LIN {X 0,Y 525.13,Z 398.918,A -85,B 0,C 180,E1 -4783.003,E2 -4783.003} C_VEL
LIN {X 0,Y 525.379,Z 385.467,A -85,B 0,C 180,E1 -4783.44,E2 -4783.44} C_VEL
LIN {X 0,Y 525.572,Z 372.166,A -85,B 0,C 180,E1 -4783.706,E2 -4783.706} C_VEL
LIN {X 0,Y 525.827,Z 279.836,A -85,B 0,C 180,E1 -4784.974,E2 -4784.974} C_VEL
LIN {X 0,Y 524.249,Z 269.867,A -85,B 0,C 180,E1 -4785.172,E2 -4785.172} C_VEL
LIN {X 0,Y 524.68,Z 249.874,A -85,B 0,C 180,E1 -4788.307,E2 -4788.307} C_VEL
LIN {X 0,Y 525.077,Z 230.49,A -85,B 0,C 180,E1 -4791.391,E2 -4791.391} C_VEL
LIN {X 0,Y 525.279,Z 221.566,A -85,B 0,C 180,E1 -4792.831,E2 -4792.831} C_VEL
LIN {X 0,Y 523.919,Z 214.225,A -85,B 0,C 180,E1 -4794.108,E2 -4794.108} C_VEL
LIN {X 0,Y 523.925,Z 214.226,A -85,B 0,C 180,E1 -4797.134,E2 -4797.134} C_VEL
LIN {X 0,Y 523.939,Z 214.222,A -85,B 0,C 180,E1 -4799.756,E2 -4799.756} C_VEL
LIN {X 0,Y 523.935,Z 214.217,A -85,B 0,C 180,E1 -4802.449,E2 -4802.449} C_VEL
LIN {X 0,Y 523.919,Z 214.224,A -85,B 0,C 180,E1 -4805.227,E2 -4805.227} C_VEL
LIN {X 0,Y 523.914,Z 214.221,A -85,B 0,C 180,E1 -4808.102,E2 -4808.102} C_VEL
LIN {X 0,Y 523.938,Z 214.22,A -85,B 0,C 180,E1 -4811.092,E2 -4811.092} C_VEL
LIN {X 0,Y 523.93,Z 214.218,A -85,B 0,C 180,E1 -4814.229,E2 -4814.229} C_VEL
LIN {X 0,Y 523.893,Z 214.223,A -85,B 0,C 180,E1 -4816.83,E2 -4816.83} C_VEL
LIN {X 0,Y 523.938,Z 214.218,A -85,B 0,C 180,E1 -4818.907,E2 -4818.907} C_VEL
LIN {X 0,Y 523.913,Z 214.221,A -85,B 0,C 180,E1 -4821.898,E2 -4821.898} C_VEL
LIN {X 0,Y 523.922,Z 214.22,A -85,B 0,C 180,E1 -4824.912,E2 -4824.912} C_VEL
LIN {X 0,Y 523.936,Z 214.222,A -85,B 0,C 180,E1 -4827.68,E2 -4827.68} C_VEL
LIN {X 0,Y 523.954,Z 214.212,A -85,B 0,C 180,E1 -4830.677,E2 -4830.677} C_VEL
LIN {X 0,Y 523.938,Z 214.219,A -85,B 0,C 180,E1 -4833.727,E2 -4833.727} C_VEL
LIN {X 0,Y 523.913,Z 214.219,A -85,B 0,C 180,E1 -4836.27,E2 -4836.27} C_VEL
LIN {X 0,Y 523.946,Z 214.214,A -85,B 0,C 180,E1 -4838.767,E2 -4838.767} C_VEL
LIN {X 0,Y 523.948,Z 214.221,A -85,B 0,C 180,E1 -4841.221,E2 -4841.221} C_VEL
LIN {X 0,Y 523.928,Z 214.223,A -85,B 0,C 180,E1 -4843.639,E2 -4843.639} C_VEL
LIN {X 0,Y 523.944,Z 214.216,A -85,B 0,C 180,E1 -4846.028,E2 -4846.028} C_VEL
LIN {X 0,Y 523.995,Z 214.212,A -85,B 0,C 180,E1 -4849.177,E2 -4849.177} C_VEL
LIN {X 0,Y 524.029,Z 214.203,A -85,B 0,C 180,E1 -4852.293,E2 -4852.293} C_VEL
LIN {X 0,Y 524.079,Z 214.198,A -85,B 0,C 180,E1 -4854.614,E2 -4854.614} C_VEL
LIN {X 0,Y 524.112,Z 214.197,A -85,B 0,C 180,E1 -4857.695,E2 -4857.695} C_VEL
LIN {X 0,Y 524.119,Z 214.194,A -85,B 0,C 180,E1 -4860.768,E2 -4860.768} C_VEL
LIN {X 0,Y 524.041,Z 214.205,A -85,B 0,C 180,E1 -4863.075,E2 -4863.075} C_VEL
LIN {X 0,Y 524.033,Z 214.204,A -85,B 0,C 180,E1 -4866.159,E2 -4866.159} C_VEL
LIN {X 0,Y 523.985,Z 214.214,A -85,B 0,C 180,E1 -4869.262,E2 -4869.262} C_VEL
LIN {X 0,Y 524.001,Z 214.211,A -85,B 0,C 180,E1 -4871.737,E2 -4871.737} C_VEL
LIN {X 0,Y 523.988,Z 214.212,A -85,B 0,C 180,E1 -4875.05,E2 -4875.05} C_VEL
LIN {X 0,Y 523.946,Z 214.214,A -85,B 0,C 180,E1 -4877.97,E2 -4877.97} C_VEL
LIN {X 0,Y 523.959,Z 214.213,A -85,B 0,C 180,E1 -4880.411,E2 -4880.411} C_VEL
LIN {X 0,Y 523.911,Z 214.219,A -85,B 0,C 180,E1 -4882.894,E2 -4882.894} C_VEL
LIN {X 0,Y 523.911,Z 214.227,A -85,B 0,C 180,E1 -4885.421,E2 -4885.421} C_VEL
LIN {X 0,Y 523.957,Z 214.215,A -85,B 0,C 180,E1 -4888,E2 -4888} C_VEL
LIN {X 0,Y 523.941,Z 214.216,A -85,B 0,C 180,E1 -4890.854,E2 -4890.854} C_VEL
LIN {X 0,Y 523.961,Z 214.218,A -85,B 0,C 180,E1 -4893.734,E2 -4893.734} C_VEL
LIN {X 0,Y 523.9,Z 214.219,A -85,B 0,C 180,E1 -4896.401,E2 -4896.401} C_VEL
LIN {X 0,Y 523.921,Z 214.223,A -85,B 0,C 180,E1 -4899.085,E2 -4899.085} C_VEL
LIN {X 0,Y 523.945,Z 214.216,A -85,B 0,C 180,E1 -4902.12,E2 -4902.12} C_VEL
LIN {X 0,Y 523.94,Z 214.225,A -85,B 0,C 180,E1 -4905.311,E2 -4905.311} C_VEL
LIN {X 0,Y 523.893,Z 214.222,A -85,B 0,C 180,E1 -4906.884,E2 -4906.884} C_VEL
LIN {X 0,Y 523.226,Z 214.314,A -85,B 0,C 180,E1 -4907.526,E2 -4907.526} C_VEL
LIN {X 0,Y 520.369,Z 214.665,A -85,B 0,C 180,E1 -4908.568,E2 -4908.568} C_VEL
LIN {X 0,Y 517.964,Z 214.969,A -85,B 0,C 180,E1 -4909.407,E2 -4909.407} C_VEL
LIN {X 0,Y 516.948,Z 215.089,A -85,B 0,C 180,E1 -4910.055,E2 -4910.055} C_VEL
LIN {X 0,Y 516.873,Z 215.097,A -85,B 0,C 180,E1 -4910.274,E2 -4910.274} C_VEL
LIN {X 0,Y 516.877,Z 215.106,A -85,B 0,C 180,E1 -4913.344,E2 -4913.344} C_VEL
LIN {X 0,Y 516.887,Z 215.096,A -85,B 0,C 180,E1 -4916.119,E2 -4916.119} C_VEL
LIN {X 0,Y 516.894,Z 215.097,A -85,B 0,C 180,E1 -4918.936,E2 -4918.936} C_VEL
LIN {X 0,Y 516.865,Z 215.102,A -85,B 0,C 180,E1 -4921.582,E2 -4921.582} C_VEL
LIN {X 0,Y 516.961,Z 215.274,A -85,B 0,C 180,E1 -4923.533,E2 -4923.533} C_VEL
LIN {X 0,Y 517.58,Z 220.097,A -85,B 0,C 180,E1 -4924.461,E2 -4924.461} C_VEL
LIN {X 0,Y 517.327,Z 236.48,A -85,B 0,C 180,E1 -4927.488,E2 -4927.488} C_VEL
LIN {X 0,Y 517.234,Z 242.99,A -85,B 0,C 180,E1 -4928.68,E2 -4928.68} C_VEL
LIN {X 0,Y 519.15,Z 254.45,A -85,B 0,C 180,E1 -4928.909,E2 -4928.909} C_VEL
LIN {X 0,Y 518.623,Z 349.842,A -85,B 0,C 180,E1 -4930.249,E2 -4930.249} C_VEL
LIN {X 0,Y 518.444,Z 363.428,A -85,B 0,C 180,E1 -4930.602,E2 -4930.602} C_VEL
LIN {X 0,Y 518.199,Z 376.588,A -85,B 0,C 180,E1 -4931.117,E2 -4931.117} C_VEL
LIN {X 0,Y 517.949,Z 388.728,A -85,B 0,C 180,E1 -4931.774,E2 -4931.774} C_VEL
LIN {X 0,Y 517.563,Z 400.832,A -85,B 0,C 180,E1 -4932.618,E2 -4932.618} C_VEL
LIN {X 0,Y 517.292,Z 411.073,A -85,B 0,C 180,E1 -4933.524,E2 -4933.524} C_VEL
LIN {X 0,Y 517.046,Z 419.545,A -85,B 0,C 180,E1 -4934.44,E2 -4934.44} C_VEL
LIN {X 0,Y 516.757,Z 428.512,A -85,B 0,C 180,E1 -4935.629,E2 -4935.629} C_VEL
LIN {X 0,Y 516.583,Z 435.771,A -85,B 0,C 180,E1 -4936.828,E2 -4936.828} C_VEL
LIN {X 0,Y 516.486,Z 440.64,A -85,B 0,C 180,E1 -4937.824,E2 -4937.824} C_VEL
LIN {X 0,Y 516.377,Z 445.343,A -85,B 0,C 180,E1 -4939.016,E2 -4939.016} C_VEL
LIN {X 0,Y 516.282,Z 448.91,A -85,B 0,C 180,E1 -4940.203,E2 -4940.203} C_VEL
LIN {X 0,Y 516.234,Z 451.446,A -85,B 0,C 180,E1 -4941.387,E2 -4941.387} C_VEL
LIN {X 0,Y 516.254,Z 452.623,A -85,B 0,C 180,E1 -4942.176,E2 -4942.176} C_VEL
LIN {X 0,Y 516.273,Z 453.665,A -85,B 0,C 180,E1 -4943.591,E2 -4943.591} C_VEL
LIN {X 0,Y 516.273,Z 453.657,A -85,B 0,C 180,E1 -4944.532,E2 -4944.532} C_VEL
LIN {X 0,Y 516.217,Z 453.229,A -85,B 0,C 180,E1 -4945.314,E2 -4945.314} C_VEL
LIN {X 0,Y 516.304,Z 452.364,A -85,B 0,C 180,E1 -4946.097,E2 -4946.097} C_VEL
LIN {X 0,Y 516.295,Z 451.11,A -85,B 0,C 180,E1 -4946.879,E2 -4946.879} C_VEL
LIN {X 0,Y 516.311,Z 448.459,A -85,B 0,C 180,E1 -4948.05,E2 -4948.05} C_VEL
LIN {X 0,Y 516.283,Z 444.815,A -85,B 0,C 180,E1 -4949.22,E2 -4949.22} C_VEL
LIN {X 0,Y 516.453,Z 440.065,A -85,B 0,C 180,E1 -4950.39,E2 -4950.39} C_VEL
LIN {X 0,Y 516.558,Z 434.09,A -85,B 0,C 180,E1 -4951.559,E2 -4951.559} C_VEL
LIN {X 0,Y 516.82,Z 426.665,A -85,B 0,C 180,E1 -4952.728,E2 -4952.728} C_VEL
LIN {X 0,Y 517.036,Z 419.105,A -85,B 0,C 180,E1 -4953.702,E2 -4953.702} C_VEL
LIN {X 0,Y 517.288,Z 409.943,A -85,B 0,C 180,E1 -4954.676,E2 -4954.676} C_VEL
LIN {X 0,Y 517.632,Z 399.759,A -85,B 0,C 180,E1 -4955.551,E2 -4955.551} C_VEL
LIN {X 0,Y 517.936,Z 388.496,A -85,B 0,C 180,E1 -4956.33,E2 -4956.33} C_VEL
LIN {X 0,Y 518.177,Z 376.803,A -85,B 0,C 180,E1 -4956.962,E2 -4956.962} C_VEL
LIN {X 0,Y 518.46,Z 363.864,A -85,B 0,C 180,E1 -4957.472,E2 -4957.472} C_VEL
LIN {X 0,Y 518.602,Z 351.137,A -85,B 0,C 180,E1 -4957.813,E2 -4957.813} C_VEL
LIN {X 0,Y 518.884,Z 303.338,A -85,B 0,C 180,E1 -4958.501,E2 -4958.501} C_VEL
LIN {X 0,Y 519.104,Z 253.077,A -85,B 0,C 180,E1 -4959.201,E2 -4959.201} C_VEL
LIN {X 0,Y 517.252,Z 243.013,A -85,B 0,C 180,E1 -4959.408,E2 -4959.408} C_VEL
LIN {X 0,Y 517.52,Z 228.477,A -85,B 0,C 180,E1 -4962.102,E2 -4962.102} C_VEL
LIN {X 0,Y 517.546,Z 218.647,A -85,B 0,C 180,E1 -4963.948,E2 -4963.948} C_VEL
LIN {X 0,Y 516.993,Z 215.091,A -85,B 0,C 180,E1 -4964.666,E2 -4964.666} C_VEL
LIN {X 0,Y 516.905,Z 215.095,A -85,B 0,C 180,E1 -4967.871,E2 -4967.871} C_VEL
LIN {X 0,Y 516.916,Z 215.1,A -85,B 0,C 180,E1 -4970.701,E2 -4970.701} C_VEL
LIN {X 0,Y 516.906,Z 215.093,A -85,B 0,C 180,E1 -4974.072,E2 -4974.072} C_VEL
LIN {X 0,Y 516.9,Z 215.101,A -85,B 0,C 180,E1 -4976.659,E2 -4976.659} C_VEL
LIN {X 0,Y 516.913,Z 215.091,A -85,B 0,C 180,E1 -4979.523,E2 -4979.523} C_VEL
LIN {X 0,Y 516.898,Z 215.1,A -85,B 0,C 180,E1 -4982.543,E2 -4982.543} C_VEL
LIN {X 0,Y 516.866,Z 215.098,A -85,B 0,C 180,E1 -4985.329,E2 -4985.329} C_VEL
LIN {X 0,Y 516.881,Z 215.095,A -85,B 0,C 180,E1 -4987.943,E2 -4987.943} C_VEL
LIN {X 0,Y 516.885,Z 215.103,A -85,B 0,C 180,E1 -4990.742,E2 -4990.742} C_VEL
LIN {X 0,Y 516.884,Z 215.101,A -85,B 0,C 180,E1 -4992.831,E2 -4992.831} C_VEL
LIN {X 0,Y 516.897,Z 215.097,A -85,B 0,C 180,E1 -4995.007,E2 -4995.007} C_VEL
LIN {X 0,Y 516.912,Z 215.096,A -85,B 0,C 180,E1 -4998.399,E2 -4998.399} C_VEL
LIN {X 0,Y 516.881,Z 215.096,A -85,B 0,C 180,E1 -5001.284,E2 -5001.284} C_VEL
LIN {X 0,Y 516.869,Z 215.099,A -85,B 0,C 180,E1 -5004.219,E2 -5004.219} C_VEL
LIN {X 0,Y 516.896,Z 215.096,A -85,B 0,C 180,E1 -5007.053,E2 -5007.053} C_VEL
LIN {X 0,Y 516.893,Z 215.093,A -85,B 0,C 180,E1 -5009.796,E2 -5009.796} C_VEL
LIN {X 0,Y 516.922,Z 215.096,A -85,B 0,C 180,E1 -5012.467,E2 -5012.467} C_VEL
LIN {X 0,Y 516.877,Z 215.095,A -85,B 0,C 180,E1 -5015.644,E2 -5015.644} C_VEL
LIN {X 0,Y 516.887,Z 215.101,A -85,B 0,C 180,E1 -5018.462,E2 -5018.462} C_VEL
LIN {X 0,Y 516.895,Z 215.097,A -85,B 0,C 180,E1 -5020.954,E2 -5020.954} C_VEL
LIN {X 0,Y 516.901,Z 215.092,A -85,B 0,C 180,E1 -5023.41,E2 -5023.41} C_VEL
LIN {X 0,Y 516.885,Z 215.094,A -85,B 0,C 180,E1 -5025.833,E2 -5025.833} C_VEL
LIN {X 0,Y 516.951,Z 215.089,A -85,B 0,C 180,E1 -5029.028,E2 -5029.028} C_VEL
LIN {X 0,Y 516.963,Z 215.087,A -85,B 0,C 180,E1 -5032.186,E2 -5032.186} C_VEL
LIN {X 0,Y 517.025,Z 215.085,A -85,B 0,C 180,E1 -5034.54,E2 -5034.54} C_VEL
LIN {X 0,Y 517.083,Z 215.069,A -85,B 0,C 180,E1 -5037.663,E2 -5037.663} C_VEL
LIN {X 0,Y 517.093,Z 215.075,A -85,B 0,C 180,E1 -5040.779,E2 -5040.779} C_VEL
LIN {X 0,Y 516.985,Z 215.084,A -85,B 0,C 180,E1 -5043.117,E2 -5043.117} C_VEL
LIN {X 0,Y 517.009,Z 215.083,A -85,B 0,C 180,E1 -5046.243,E2 -5046.243} C_VEL
LIN {X 0,Y 516.943,Z 215.087,A -85,B 0,C 180,E1 -5049.389,E2 -5049.389} C_VEL
LIN {X 0,Y 516.953,Z 215.086,A -85,B 0,C 180,E1 -5051.807,E2 -5051.807} C_VEL
LIN {X 0,Y 516.948,Z 215.088,A -85,B 0,C 180,E1 -5055.148,E2 -5055.148} C_VEL
LIN {X 0,Y 516.916,Z 215.094,A -85,B 0,C 180,E1 -5058.223,E2 -5058.223} C_VEL
LIN {X 0,Y 516.913,Z 215.098,A -85,B 0,C 180,E1 -5060.701,E2 -5060.701} C_VEL
LIN {X 0,Y 516.903,Z 215.094,A -85,B 0,C 180,E1 -5064.072,E2 -5064.072} C_VEL
LIN {X 0,Y 516.897,Z 215.101,A -85,B 0,C 180,E1 -5066.659,E2 -5066.659} C_VEL
LIN {X 0,Y 516.91,Z 215.091,A -85,B 0,C 180,E1 -5069.523,E2 -5069.523} C_VEL
LIN {X 0,Y 516.895,Z 215.102,A -85,B 0,C 180,E1 -5072.543,E2 -5072.543} C_VEL
LIN {X 0,Y 516.864,Z 215.097,A -85,B 0,C 180,E1 -5075.329,E2 -5075.329} C_VEL
LIN {X 0,Y 516.879,Z 215.096,A -85,B 0,C 180,E1 -5077.943,E2 -5077.943} C_VEL
LIN {X 0,Y 516.882,Z 215.101,A -85,B 0,C 180,E1 -5080.742,E2 -5080.742} C_VEL
LIN {X 0,Y 516.881,Z 215.096,A -85,B 0,C 180,E1 -5083.903,E2 -5083.903} C_VEL
LIN {X 0,Y 516.882,Z 215.098,A -85,B 0,C 180,E1 -5086.107,E2 -5086.107} C_VEL
LIN {X 0,Y 516.883,Z 215.095,A -85,B 0,C 180,E1 -5089.258,E2 -5089.258} C_VEL
LIN {X 0,Y 516.861,Z 215.102,A -85,B 0,C 180,E1 -5092.274,E2 -5092.274} C_VEL
LIN {X 0,Y 516.883,Z 215.096,A -85,B 0,C 180,E1 -5095.175,E2 -5095.175} C_VEL
LIN {X 0,Y 516.875,Z 215.097,A -85,B 0,C 180,E1 -5097.975,E2 -5097.975} C_VEL
LIN {X 0,Y 516.922,Z 215.097,A -85,B 0,C 180,E1 -5100.696,E2 -5100.696} C_VEL
LIN {X 0,Y 516.905,Z 215.095,A -85,B 0,C 180,E1 -5103.341,E2 -5103.341} C_VEL
LIN {X 0,Y 516.908,Z 215.177,A -85,B 0,C 180,E1 -5105.752,E2 -5105.752} C_VEL
LIN {X 0,Y 518.35,Z 223.667,A -85,B 0,C 180,E1 -5107.217,E2 -5107.217} C_VEL
LIN {X 0,Y 517.938,Z 240.677,A -85,B 0,C 180,E1 -5109.979,E2 -5109.979} C_VEL
LIN {X 0,Y 517.486,Z 258.383,A -85,B 0,C 180,E1 -5112.819,E2 -5112.819} C_VEL
LIN {X 0,Y 517.275,Z 269.968,A -85,B 0,C 180,E1 -5114.636,E2 -5114.636} C_VEL
LIN {X 0,Y 519.06,Z 282.453,A -85,B 0,C 180,E1 -5114.865,E2 -5114.865} C_VEL
LIN {X 0,Y 518.609,Z 377.87,A -85,B 0,C 180,E1 -5116.206,E2 -5116.206} C_VEL
LIN {X 0,Y 518.373,Z 391.174,A -85,B 0,C 180,E1 -5116.55,E2 -5116.55} C_VEL
LIN {X 0,Y 518.092,Z 403.355,A -85,B 0,C 180,E1 -5117.016,E2 -5117.016} C_VEL
LIN {X 0,Y 517.768,Z 415.713,A -85,B 0,C 180,E1 -5117.66,E2 -5117.66} C_VEL
LIN {X 0,Y 517.554,Z 427.254,A -85,B 0,C 180,E1 -5118.446,E2 -5118.446} C_VEL
LIN {X 0,Y 517.22,Z 437.703,A -85,B 0,C 180,E1 -5119.331,E2 -5119.331} C_VEL
LIN {X 0,Y 516.95,Z 446.247,A -85,B 0,C 180,E1 -5120.216,E2 -5120.216} C_VEL
LIN {X 0,Y 516.724,Z 454.13,A -85,B 0,C 180,E1 -5121.199,E2 -5121.199} C_VEL
LIN {X 0,Y 516.536,Z 461.829,A -85,B 0,C 180,E1 -5122.377,E2 -5122.377} C_VEL
LIN {X 0,Y 516.39,Z 468.926,A -85,B 0,C 180,E1 -5123.749,E2 -5123.749} C_VEL
LIN {X 0,Y 516.313,Z 473.647,A -85,B 0,C 180,E1 -5124.924,E2 -5124.924} C_VEL
LIN {X 0,Y 516.352,Z 477.256,A -85,B 0,C 180,E1 -5126.098,E2 -5126.098} C_VEL
LIN {X 0,Y 516.282,Z 479.114,A -85,B 0,C 180,E1 -5126.879,E2 -5126.879} C_VEL
LIN {X 0,Y 516.261,Z 480.509,A -85,B 0,C 180,E1 -5127.659,E2 -5127.659} C_VEL
LIN {X 0,Y 516.161,Z 482.109,A -85,B 0,C 180,E1 -5129.22,E2 -5129.22} C_VEL
LIN {X 0,Y 516.157,Z 482.324,A -85,B 0,C 180,E1 -5130,E2 -5130} C_VEL
LIN {X 0,Y 516.192,Z 481.502,A -85,B 0,C 180,E1 -5131.56,E2 -5131.56} C_VEL
LIN {X 0,Y 516.261,Z 480.508,A -85,B 0,C 180,E1 -5132.341,E2 -5132.341} C_VEL
LIN {X 0,Y 516.282,Z 479.113,A -85,B 0,C 180,E1 -5133.121,E2 -5133.121} C_VEL
LIN {X 0,Y 516.311,Z 476.179,A -85,B 0,C 180,E1 -5134.294,E2 -5134.294} C_VEL
LIN {X 0,Y 516.374,Z 472.206,A -85,B 0,C 180,E1 -5135.467,E2 -5135.467} C_VEL
LIN {X 0,Y 516.422,Z 467.014,A -85,B 0,C 180,E1 -5136.659,E2 -5136.659} C_VEL
LIN {X 0,Y 516.575,Z 460.656,A -85,B 0,C 180,E1 -5137.819,E2 -5137.819} C_VEL
LIN {X 0,Y 516.769,Z 452.625,A -85,B 0,C 180,E1 -5138.998,E2 -5138.998} C_VEL
LIN {X 0,Y 516.98,Z 444.442,A -85,B 0,C 180,E1 -5139.981,E2 -5139.981} C_VEL
LIN {X 0,Y 517.331,Z 434.466,A -85,B 0,C 180,E1 -5140.964,E2 -5140.964} C_VEL
LIN {X 0,Y 517.604,Z 424.623,A -85,B 0,C 180,E1 -5141.752,E2 -5141.752} C_VEL
LIN {X 0,Y 517.849,Z 413.514,A -85,B 0,C 180,E1 -5142.465,E2 -5142.465} C_VEL
LIN {X 0,Y 518.132,Z 401.058,A -85,B 0,C 180,E1 -5143.082,E2 -5143.082} C_VEL
LIN {X 0,Y 518.442,Z 388.005,A -85,B 0,C 180,E1 -5143.548,E2 -5143.548} C_VEL
LIN {X 0,Y 518.629,Z 374.978,A -85,B 0,C 180,E1 -5143.843,E2 -5143.843} C_VEL
LIN {X 0,Y 518.989,Z 280.748,A -85,B 0,C 180,E1 -5145.16,E2 -5145.16} C_VEL
LIN {X 0,Y 517.238,Z 269.601,A -85,B 0,C 180,E1 -5145.393,E2 -5145.393} C_VEL
LIN {X 0,Y 517.721,Z 249.417,A -85,B 0,C 180,E1 -5148.603,E2 -5148.603} C_VEL
LIN {X 0,Y 518.132,Z 231.593,A -85,B 0,C 180,E1 -5151.483,E2 -5151.483} C_VEL
LIN {X 0,Y 518.327,Z 222.878,A -85,B 0,C 180,E1 -5152.912,E2 -5152.912} C_VEL
LIN {X 0,Y 516.899,Z 215.098,A -85,B 0,C 180,E1 -5154.314,E2 -5154.314} C_VEL
LIN {X 0,Y 516.901,Z 215.102,A -85,B 0,C 180,E1 -5157.534,E2 -5157.534} C_VEL
LIN {X 0,Y 516.888,Z 215.096,A -85,B 0,C 180,E1 -5160.204,E2 -5160.204} C_VEL
LIN {X 0,Y 516.897,Z 215.096,A -85,B 0,C 180,E1 -5162.947,E2 -5162.947} C_VEL
LIN {X 0,Y 516.869,Z 215.102,A -85,B 0,C 180,E1 -5165.781,E2 -5165.781} C_VEL
LIN {X 0,Y 516.88,Z 215.096,A -85,B 0,C 180,E1 -5168.716,E2 -5168.716} C_VEL
LIN {X 0,Y 516.908,Z 215.097,A -85,B 0,C 180,E1 -5171.776,E2 -5171.776} C_VEL
LIN {X 0,Y 516.896,Z 215.096,A -85,B 0,C 180,E1 -5175.007,E2 -5175.007} C_VEL
LIN {X 0,Y 516.91,Z 215.092,A -85,B 0,C 180,E1 -5178.399,E2 -5178.399} C_VEL
LIN {X 0,Y 516.877,Z 215.102,A -85,B 0,C 180,E1 -5181.284,E2 -5181.284} C_VEL
LIN {X 0,Y 516.867,Z 215.097,A -85,B 0,C 180,E1 -5184.219,E2 -5184.219} C_VEL
LIN {X 0,Y 516.882,Z 215.096,A -85,B 0,C 180,E1 -5187.052,E2 -5187.052} C_VEL
LIN {X 0,Y 516.892,Z 215.095,A -85,B 0,C 180,E1 -5189.796,E2 -5189.796} C_VEL
LIN {X 0,Y 516.898,Z 215.093,A -85,B 0,C 180,E1 -5192.466,E2 -5192.466} C_VEL
LIN {X 0,Y 516.867,Z 215.098,A -85,B 0,C 180,E1 -5195.07,E2 -5195.07} C_VEL
LIN {X 0,Y 516.87,Z 215.101,A -85,B 0,C 180,E1 -5197.622,E2 -5197.622} C_VEL
LIN {X 0,Y 516.932,Z 215.089,A -85,B 0,C 180,E1 -5200.13,E2 -5200.13} C_VEL
LIN {X 0,Y 516.906,Z 215.091,A -85,B 0,C 180,E1 -5202.595,E2 -5202.595} C_VEL
LIN {X 0,Y 516.953,Z 215.089,A -85,B 0,C 180,E1 -5205.03,E2 -5205.03} C_VEL
LIN {X 0,Y 516.967,Z 215.082,A -85,B 0,C 180,E1 -5208.234,E2 -5208.234} C_VEL
LIN {X 0,Y 516.965,Z 215.093,A -85,B 0,C 180,E1 -5211.4,E2 -5211.4} C_VEL
LIN {X 0,Y 517.009,Z 215.083,A -85,B 0,C 180,E1 -5213.757,E2 -5213.757} C_VEL
LIN {X 0,Y 517.082,Z 215.073,A -85,B 0,C 180,E1 -5217.663,E2 -5217.663} C_VEL
LIN {X 0,Y 517.09,Z 215.07,A -85,B 0,C 180,E1 -5220.779,E2 -5220.779} C_VEL
LIN {X 0,Y 516.984,Z 215.085,A -85,B 0,C 180,E1 -5223.117,E2 -5223.117} C_VEL
LIN {X 0,Y 516.995,Z 215.081,A -85,B 0,C 180,E1 -5226.243,E2 -5226.243} C_VEL
LIN {X 0,Y 516.941,Z 215.093,A -85,B 0,C 180,E1 -5229.39,E2 -5229.39} C_VEL
LIN {X 0,Y 516.953,Z 215.088,A -85,B 0,C 180,E1 -5231.807,E2 -5231.807} C_VEL
LIN {X 0,Y 516.94,Z 215.091,A -85,B 0,C 180,E1 -5235.144,E2 -5235.144} C_VEL
LIN {X 0,Y 516.914,Z 215.088,A -85,B 0,C 180,E1 -5238.223,E2 -5238.223} C_VEL
LIN {X 0,Y 516.906,Z 215.092,A -85,B 0,C 180,E1 -5240.702,E2 -5240.702} C_VEL
LIN {X 0,Y 516.887,Z 215.095,A -85,B 0,C 180,E1 -5244.073,E2 -5244.073} C_VEL
LIN {X 0,Y 516.905,Z 215.09,A -85,B 0,C 180,E1 -5246.659,E2 -5246.659} C_VEL
LIN {X 0,Y 516.91,Z 215.097,A -85,B 0,C 180,E1 -5249.523,E2 -5249.523} C_VEL
LIN {X 0,Y 516.897,Z 215.093,A -85,B 0,C 180,E1 -5252.543,E2 -5252.543} C_VEL
LIN {X 0,Y 516.866,Z 215.105,A -85,B 0,C 180,E1 -5255.329,E2 -5255.329} C_VEL
LIN {X 0,Y 516.88,Z 215.097,A -85,B 0,C 180,E1 -5257.943,E2 -5257.943} C_VEL
LIN {X 0,Y 516.884,Z 215.096,A -85,B 0,C 180,E1 -5260.742,E2 -5260.742} C_VEL
LIN {X 0,Y 516.883,Z 215.098,A -85,B 0,C 180,E1 -5263.903,E2 -5263.903} C_VEL
LIN {X 0,Y 516.846,Z 215.1,A -85,B 0,C 180,E1 -5266.886,E2 -5266.886} C_VEL
LIN {X 0,Y 516.886,Z 215.101,A -85,B 0,C 180,E1 -5269.59,E2 -5269.59} C_VEL
LIN {X 0,Y 516.873,Z 215.097,A -85,B 0,C 180,E1 -5270.274,E2 -5270.274} C_VEL
LIN {X 0,Y 516.232,Z 215.18,A -85,B 0,C 180,E1 -5270.924,E2 -5270.924} C_VEL
LIN {X 0,Y 513.391,Z 215.54,A -85,B 0,C 180,E1 -5271.98,E2 -5271.98} C_VEL
LIN {X 0,Y 510.967,Z 215.845,A -85,B 0,C 180,E1 -5272.83,E2 -5272.83} C_VEL
LIN {X 0,Y 509.913,Z 215.973,A -85,B 0,C 180,E1 -5273.487,E2 -5273.487} C_VEL
LIN {X 0,Y 509.822,Z 215.982,A -85,B 0,C 180,E1 -5273.709,E2 -5273.709} C_VEL
LIN {X 0,Y 509.844,Z 215.973,A -85,B 0,C 180,E1 -5276.538,E2 -5276.538} C_VEL
LIN {X 0,Y 509.848,Z 215.978,A -85,B 0,C 180,E1 -5279.334,E2 -5279.334} C_VEL
LIN {X 0,Y 509.851,Z 215.974,A -85,B 0,C 180,E1 -5282.052,E2 -5282.052} C_VEL
LIN {X 0,Y 509.904,Z 216.009,A -85,B 0,C 180,E1 -5283.361,E2 -5283.361} C_VEL
LIN {X 0,Y 510.626,Z 221.981,A -85,B 0,C 180,E1 -5284.525,E2 -5284.525} C_VEL
LIN {X 0,Y 510.333,Z 238.095,A -85,B 0,C 180,E1 -5287.533,E2 -5287.533} C_VEL
LIN {X 0,Y 510.273,Z 243.432,A -85,B 0,C 180,E1 -5288.477,E2 -5288.477} C_VEL
LIN {X 0,Y 512.315,Z 255.262,A -85,B 0,C 180,E1 -5288.711,E2 -5288.711} C_VEL
LIN {X 0,Y 511.732,Z 350.795,A -85,B 0,C 180,E1 -5290.076,E2 -5290.076} C_VEL
LIN {X 0,Y 511.546,Z 364.127,A -85,B 0,C 180,E1 -5290.435,E2 -5290.435} C_VEL
LIN {X 0,Y 511.293,Z 376.918,A -85,B 0,C 180,E1 -5290.946,E2 -5290.946} C_VEL
LIN {X 0,Y 511.017,Z 389.089,A -85,B 0,C 180,E1 -5291.615,E2 -5291.615} C_VEL
LIN {X 0,Y 510.643,Z 399.924,A -85,B 0,C 180,E1 -5292.375,E2 -5292.375} C_VEL
LIN {X 0,Y 510.358,Z 410.422,A -85,B 0,C 180,E1 -5293.294,E2 -5293.294} C_VEL
LIN {X 0,Y 510.047,Z 418.946,A -85,B 0,C 180,E1 -5294.209,E2 -5294.209} C_VEL
LIN {X 0,Y 509.742,Z 428.132,A -85,B 0,C 180,E1 -5295.427,E2 -5295.427} C_VEL
LIN {X 0,Y 509.524,Z 435.499,A -85,B 0,C 180,E1 -5296.642,E2 -5296.642} C_VEL
LIN {X 0,Y 509.417,Z 440.453,A -85,B 0,C 180,E1 -5297.652,E2 -5297.652} C_VEL
LIN {X 0,Y 509.325,Z 445.239,A -85,B 0,C 180,E1 -5298.861,E2 -5298.861} C_VEL
LIN {X 0,Y 509.222,Z 448.882,A -85,B 0,C 180,E1 -5300.066,E2 -5300.066} C_VEL
LIN {X 0,Y 509.145,Z 451.49,A -85,B 0,C 180,E1 -5301.266,E2 -5301.266} C_VEL
LIN {X 0,Y 509.163,Z 452.712,A -85,B 0,C 180,E1 -5302.066,E2 -5302.066} C_VEL
LIN {X 0,Y 509.2,Z 453.5,A -85,B 0,C 180,E1 -5302.864,E2 -5302.864} C_VEL
LIN {X 0,Y 509.182,Z 453.87,A -85,B 0,C 180,E1 -5304.456,E2 -5304.456} C_VEL
LIN {X 0,Y 509.133,Z 453.484,A -85,B 0,C 180,E1 -5305.249,E2 -5305.249} C_VEL
LIN {X 0,Y 509.198,Z 452.677,A -85,B 0,C 180,E1 -5306.043,E2 -5306.043} C_VEL
LIN {X 0,Y 509.209,Z 451.457,A -85,B 0,C 180,E1 -5306.835,E2 -5306.835} C_VEL
LIN {X 0,Y 509.22,Z 448.876,A -85,B 0,C 180,E1 -5308.023,E2 -5308.023} C_VEL
LIN {X 0,Y 509.199,Z 445.306,A -85,B 0,C 180,E1 -5309.209,E2 -5309.209} C_VEL
LIN {X 0,Y 509.371,Z 440.636,A -85,B 0,C 180,E1 -5310.395,E2 -5310.395} C_VEL
LIN {X 0,Y 509.493,Z 434.747,A -85,B 0,C 180,E1 -5311.581,E2 -5311.581} C_VEL
LIN {X 0,Y 509.667,Z 428.764,A -85,B 0,C 180,E1 -5312.569,E2 -5312.569} C_VEL
LIN {X 0,Y 509.981,Z 419.975,A -85,B 0,C 180,E1 -5313.753,E2 -5313.753} C_VEL
LIN {X 0,Y 510.272,Z 410.978,A -85,B 0,C 180,E1 -5314.74,E2 -5314.74} C_VEL
LIN {X 0,Y 510.619,Z 401.022,A -85,B 0,C 180,E1 -5315.628,E2 -5315.628} C_VEL
LIN {X 0,Y 510.97,Z 389.991,A -85,B 0,C 180,E1 -5316.416,E2 -5316.416} C_VEL
LIN {X 0,Y 511.258,Z 377.66,A -85,B 0,C 180,E1 -5317.107,E2 -5317.107} C_VEL
LIN {X 0,Y 511.548,Z 365.063,A -85,B 0,C 180,E1 -5317.624,E2 -5317.624} C_VEL
LIN {X 0,Y 511.743,Z 351.073,A -85,B 0,C 180,E1 -5318.007,E2 -5318.007} C_VEL
LIN {X 0,Y 512.208,Z 271.294,A -85,B 0,C 180,E1 -5319.153,E2 -5319.153} C_VEL
LIN {X 0,Y 512.169,Z 253.423,A -85,B 0,C 180,E1 -5319.409,E2 -5319.409} C_VEL
LIN {X 0,Y 510.23,Z 243.085,A -85,B 0,C 180,E1 -5319.639,E2 -5319.639} C_VEL
LIN {X 0,Y 510.519,Z 229.373,A -85,B 0,C 180,E1 -5322.199,E2 -5322.199} C_VEL
LIN {X 0,Y 510.614,Z 220.177,A -85,B 0,C 180,E1 -5323.938,E2 -5323.938} C_VEL
LIN {X 0,Y 509.942,Z 215.969,A -85,B 0,C 180,E1 -5324.772,E2 -5324.772} C_VEL
LIN {X 0,Y 509.871,Z 215.971,A -85,B 0,C 180,E1 -5327.993,E2 -5327.993} C_VEL
LIN {X 0,Y 509.89,Z 215.97,A -85,B 0,C 180,E1 -5330.401,E2 -5330.401} C_VEL
LIN {X 0,Y 509.833,Z 215.973,A -85,B 0,C 180,E1 -5333.563,E2 -5333.563} C_VEL
LIN {X 0,Y 509.882,Z 215.971,A -85,B 0,C 180,E1 -5336.371,E2 -5336.371} C_VEL
LIN {X 0,Y 509.861,Z 215.969,A -85,B 0,C 180,E1 -5339.726,E2 -5339.726} C_VEL
LIN {X 0,Y 509.876,Z 215.975,A -85,B 0,C 180,E1 -5342.774,E2 -5342.774} C_VEL
LIN {X 0,Y 509.826,Z 215.974,A -85,B 0,C 180,E1 -5345.578,E2 -5345.578} C_VEL
LIN {X 0,Y 509.851,Z 215.975,A -85,B 0,C 180,E1 -5348.338,E2 -5348.338} C_VEL
LIN {X 0,Y 509.857,Z 215.97,A -85,B 0,C 180,E1 -5351.425,E2 -5351.425} C_VEL
LIN {X 0,Y 509.841,Z 215.981,A -85,B 0,C 180,E1 -5354.67,E2 -5354.67} C_VEL
LIN {X 0,Y 509.852,Z 215.972,A -85,B 0,C 180,E1 -5358.104,E2 -5358.104} C_VEL
LIN {X 0,Y 509.847,Z 215.98,A -85,B 0,C 180,E1 -5360.647,E2 -5360.647} C_VEL
LIN {X 0,Y 509.81,Z 215.975,A -85,B 0,C 180,E1 -5363.645,E2 -5363.645} C_VEL
LIN {X 0,Y 509.86,Z 215.977,A -85,B 0,C 180,E1 -5366.539,E2 -5366.539} C_VEL
LIN {X 0,Y 509.847,Z 215.972,A -85,B 0,C 180,E1 -5369.334,E2 -5369.334} C_VEL
LIN {X 0,Y 509.884,Z 215.968,A -85,B 0,C 180,E1 -5372.054,E2 -5372.054} C_VEL
LIN {X 0,Y 509.81,Z 215.984,A -85,B 0,C 180,E1 -5374.7,E2 -5374.7} C_VEL
LIN {X 0,Y 509.827,Z 215.974,A -85,B 0,C 180,E1 -5377.458,E2 -5377.458} C_VEL
LIN {X 0,Y 509.917,Z 215.962,A -85,B 0,C 180,E1 -5379.845,E2 -5379.845} C_VEL
LIN {X 0,Y 509.868,Z 215.97,A -85,B 0,C 180,E1 -5383.174,E2 -5383.174} C_VEL
LIN {X 0,Y 509.856,Z 215.97,A -85,B 0,C 180,E1 -5385.634,E2 -5385.634} C_VEL
LIN {X 0,Y 509.913,Z 215.968,A -85,B 0,C 180,E1 -5388.874,E2 -5388.874} C_VEL
LIN {X 0,Y 509.922,Z 215.964,A -85,B 0,C 180,E1 -5392.078,E2 -5392.078} C_VEL
LIN {X 0,Y 509.976,Z 215.962,A -85,B 0,C 180,E1 -5394.464,E2 -5394.464} C_VEL
LIN {X 0,Y 510.054,Z 215.945,A -85,B 0,C 180,E1 -5397.631,E2 -5397.631} C_VEL
LIN {X 0,Y 510.063,Z 215.95,A -85,B 0,C 180,E1 -5400.789,E2 -5400.789} C_VEL
LIN {X 0,Y 509.928,Z 215.963,A -85,B 0,C 180,E1 -5403.16,E2 -5403.16} C_VEL
LIN {X 0,Y 509.977,Z 215.96,A -85,B 0,C 180,E1 -5406.33,E2 -5406.33} C_VEL
LIN {X 0,Y 509.911,Z 215.97,A -85,B 0,C 180,E1 -5408.72,E2 -5408.72} C_VEL
LIN {X 0,Y 509.905,Z 215.965,A -85,B 0,C 180,E1 -5411.932,E2 -5411.932} C_VEL
LIN {X 0,Y 509.895,Z 215.966,A -85,B 0,C 180,E1 -5415.242,E2 -5415.242} C_VEL
LIN {X 0,Y 509.861,Z 215.977,A -85,B 0,C 180,E1 -5418.484,E2 -5418.484} C_VEL
LIN {X 0,Y 509.851,Z 215.974,A -85,B 0,C 180,E1 -5421.002,E2 -5421.002} C_VEL
LIN {X 0,Y 509.858,Z 215.976,A -85,B 0,C 180,E1 -5424.427,E2 -5424.427} C_VEL
LIN {X 0,Y 509.859,Z 215.972,A -85,B 0,C 180,E1 -5427.057,E2 -5427.057} C_VEL
LIN {X 0,Y 509.858,Z 215.97,A -85,B 0,C 180,E1 -5429.751,E2 -5429.751} C_VEL
LIN {X 0,Y 509.867,Z 215.974,A -85,B 0,C 180,E1 -5432.773,E2 -5432.773} C_VEL
LIN {X 0,Y 509.823,Z 215.974,A -85,B 0,C 180,E1 -5435.578,E2 -5435.578} C_VEL
LIN {X 0,Y 509.849,Z 215.976,A -85,B 0,C 180,E1 -5438.338,E2 -5438.338} C_VEL
LIN {X 0,Y 509.853,Z 215.97,A -85,B 0,C 180,E1 -5441.426,E2 -5441.426} C_VEL
LIN {X 0,Y 509.839,Z 215.979,A -85,B 0,C 180,E1 -5444.67,E2 -5444.67} C_VEL
LIN {X 0,Y 509.851,Z 215.973,A -85,B 0,C 180,E1 -5448.104,E2 -5448.104} C_VEL
LIN {X 0,Y 509.846,Z 215.979,A -85,B 0,C 180,E1 -5450.648,E2 -5450.648} C_VEL
LIN {X 0,Y 509.81,Z 215.976,A -85,B 0,C 180,E1 -5453.646,E2 -5453.646} C_VEL
LIN {X 0,Y 509.86,Z 215.979,A -85,B 0,C 180,E1 -5456.539,E2 -5456.539} C_VEL
LIN {X 0,Y 509.844,Z 215.972,A -85,B 0,C 180,E1 -5459.334,E2 -5459.334} C_VEL
LIN {X 0,Y 509.884,Z 215.971,A -85,B 0,C 180,E1 -5462.054,E2 -5462.054} C_VEL
LIN {X 0,Y 509.81,Z 215.981,A -85,B 0,C 180,E1 -5464.7,E2 -5464.7} C_VEL
LIN {X 0,Y 509.869,Z 216.109,A -85,B 0,C 180,E1 -5465.601,E2 -5465.601} C_VEL
LIN {X 0,Y 511.38,Z 224.33,A -85,B 0,C 180,E1 -5467.043,E2 -5467.043} C_VEL
LIN {X 0,Y 510.999,Z 239.669,A -85,B 0,C 180,E1 -5469.567,E2 -5469.567} C_VEL
LIN {X 0,Y 510.536,Z 256.913,A -85,B 0,C 180,E1 -5472.371,E2 -5472.371} C_VEL
LIN {X 0,Y 510.236,Z 269.588,A -85,B 0,C 180,E1 -5474.415,E2 -5474.415} C_VEL
LIN {X 0,Y 512.148,Z 281.846,A -85,B 0,C 180,E1 -5474.65,E2 -5474.65} C_VEL
LIN {X 0,Y 511.726,Z 377.664,A -85,B 0,C 180,E1 -5476.017,E2 -5476.017} C_VEL
LIN {X 0,Y 511.477,Z 390.971,A -85,B 0,C 180,E1 -5476.365,E2 -5476.365} C_VEL
LIN {X 0,Y 511.159,Z 403.154,A -85,B 0,C 180,E1 -5476.837,E2 -5476.837} C_VEL
LIN {X 0,Y 510.872,Z 414.68,A -85,B 0,C 180,E1 -5477.439,E2 -5477.439} C_VEL
LIN {X 0,Y 510.592,Z 425.759,A -85,B 0,C 180,E1 -5478.185,E2 -5478.185} C_VEL
LIN {X 0,Y 510.266,Z 436.433,A -85,B 0,C 180,E1 -5479.083,E2 -5479.083} C_VEL
LIN {X 0,Y 509.916,Z 446.049,A -85,B 0,C 180,E1 -5480.079,E2 -5480.079} C_VEL
LIN {X 0,Y 509.672,Z 453.932,A -85,B 0,C 180,E1 -5481.076,E2 -5481.076} C_VEL
LIN {X 0,Y 509.475,Z 461.632,A -85,B 0,C 180,E1 -5482.27,E2 -5482.27} C_VEL
LIN {X 0,Y 509.308,Z 468.729,A -85,B 0,C 180,E1 -5483.662,E2 -5483.662} C_VEL
LIN {X 0,Y 509.243,Z 473.451,A -85,B 0,C 180,E1 -5484.853,E2 -5484.853} C_VEL
LIN {X 0,Y 509.245,Z 477.059,A -85,B 0,C 180,E1 -5486.043,E2 -5486.043} C_VEL
LIN {X 0,Y 509.2,Z 478.919,A -85,B 0,C 180,E1 -5486.835,E2 -5486.835} C_VEL
LIN {X 0,Y 509.19,Z 480.313,A -85,B 0,C 180,E1 -5487.627,E2 -5487.627} C_VEL
LIN {X 0,Y 509.074,Z 481.913,A -85,B 0,C 180,E1 -5489.209,E2 -5489.209} C_VEL
LIN {X 0,Y 509.068,Z 482.128,A -85,B 0,C 180,E1 -5490,E2 -5490} C_VEL
LIN {X 0,Y 509.112,Z 481.305,A -85,B 0,C 180,E1 -5491.582,E2 -5491.582} C_VEL
LIN {X 0,Y 509.19,Z 480.312,A -85,B 0,C 180,E1 -5492.373,E2 -5492.373} C_VEL
LIN {X 0,Y 509.2,Z 478.916,A -85,B 0,C 180,E1 -5493.165,E2 -5493.165} C_VEL
LIN {X 0,Y 509.203,Z 475.98,A -85,B 0,C 180,E1 -5494.354,E2 -5494.354} C_VEL
LIN {X 0,Y 509.291,Z 472.007,A -85,B 0,C 180,E1 -5495.543,E2 -5495.543} C_VEL
LIN {X 0,Y 509.4,Z 465.998,A -85,B 0,C 180,E1 -5496.914,E2 -5496.914} C_VEL
LIN {X 0,Y 509.545,Z 459.218,A -85,B 0,C 180,E1 -5498.127,E2 -5498.127} C_VEL
LIN {X 0,Y 509.748,Z 450.931,A -85,B 0,C 180,E1 -5499.323,E2 -5499.323} C_VEL
LIN {X 0,Y 510.011,Z 442.439,A -85,B 0,C 180,E1 -5500.32,E2 -5500.32} C_VEL
LIN {X 0,Y 510.382,Z 431.946,A -85,B 0,C 180,E1 -5501.316,E2 -5501.316} C_VEL
LIN {X 0,Y 510.675,Z 421.767,A -85,B 0,C 180,E1 -5502.101,E2 -5502.101} C_VEL
LIN {X 0,Y 511.022,Z 410.185,A -85,B 0,C 180,E1 -5502.813,E2 -5502.813} C_VEL
LIN {X 0,Y 511.293,Z 398.505,A -85,B 0,C 180,E1 -5503.362,E2 -5503.362} C_VEL
LIN {X 0,Y 511.57,Z 385.049,A -85,B 0,C 180,E1 -5503.81,E2 -5503.81} C_VEL
LIN {X 0,Y 511.789,Z 371.734,A -85,B 0,C 180,E1 -5504.082,E2 -5504.082} C_VEL
LIN {X 0,Y 512.108,Z 281.456,A -85,B 0,C 180,E1 -5505.356,E2 -5505.356} C_VEL
LIN {X 0,Y 510.23,Z 269.52,A -85,B 0,C 180,E1 -5505.59,E2 -5505.59} C_VEL
LIN {X 0,Y 510.726,Z 250.511,A -85,B 0,C 180,E1 -5508.659,E2 -5508.659} C_VEL
LIN {X 0,Y 511.196,Z 232.725,A -85,B 0,C 180,E1 -5511.578,E2 -5511.578} C_VEL
LIN {X 0,Y 511.412,Z 224.384,A -85,B 0,C 180,E1 -5512.966,E2 -5512.966} C_VEL
LIN {X 0,Y 509.845,Z 215.977,A -85,B 0,C 180,E1 -5514.471,E2 -5514.471} C_VEL
LIN {X 0,Y 509.86,Z 215.978,A -85,B 0,C 180,E1 -5517.057,E2 -5517.057} C_VEL
LIN {X 0,Y 509.859,Z 215.975,A -85,B 0,C 180,E1 -5519.751,E2 -5519.751} C_VEL
LIN {X 0,Y 509.875,Z 215.97,A -85,B 0,C 180,E1 -5522.774,E2 -5522.774} C_VEL
LIN {X 0,Y 509.825,Z 215.982,A -85,B 0,C 180,E1 -5525.578,E2 -5525.578} C_VEL
LIN {X 0,Y 509.85,Z 215.972,A -85,B 0,C 180,E1 -5528.338,E2 -5528.338} C_VEL
LIN {X 0,Y 509.854,Z 215.979,A -85,B 0,C 180,E1 -5531.426,E2 -5531.426} C_VEL
LIN {X 0,Y 509.84,Z 215.973,A -85,B 0,C 180,E1 -5534.67,E2 -5534.67} C_VEL
LIN {X 0,Y 509.85,Z 215.973,A -85,B 0,C 180,E1 -5538.104,E2 -5538.104} C_VEL
LIN {X 0,Y 509.839,Z 215.973,A -85,B 0,C 180,E1 -5540.647,E2 -5540.647} C_VEL
LIN {X 0,Y 509.809,Z 215.982,A -85,B 0,C 180,E1 -5543.645,E2 -5543.645} C_VEL
LIN {X 0,Y 509.842,Z 215.97,A -85,B 0,C 180,E1 -5546.538,E2 -5546.538} C_VEL
LIN {X 0,Y 509.846,Z 215.979,A -85,B 0,C 180,E1 -5549.334,E2 -5549.334} C_VEL
LIN {X 0,Y 509.849,Z 215.973,A -85,B 0,C 180,E1 -5552.052,E2 -5552.052} C_VEL
LIN {X 0,Y 509.822,Z 215.972,A -85,B 0,C 180,E1 -5554.701,E2 -5554.701} C_VEL
LIN {X 0,Y 509.827,Z 215.981,A -85,B 0,C 180,E1 -5557.458,E2 -5557.458} C_VEL
LIN {X 0,Y 509.918,Z 215.966,A -85,B 0,C 180,E1 -5559.845,E2 -5559.845} C_VEL
LIN {X 0,Y 509.872,Z 215.972,A -85,B 0,C 180,E1 -5563.174,E2 -5563.174} C_VEL
LIN {X 0,Y 509.874,Z 215.974,A -85,B 0,C 180,E1 -5565.634,E2 -5565.634} C_VEL
LIN {X 0,Y 509.913,Z 215.962,A -85,B 0,C 180,E1 -5568.875,E2 -5568.875} C_VEL
LIN {X 0,Y 509.952,Z 215.957,A -85,B 0,C 180,E1 -5572.079,E2 -5572.079} C_VEL
LIN {X 0,Y 509.979,Z 215.954,A -85,B 0,C 180,E1 -5574.464,E2 -5574.464} C_VEL
LIN {X 0,Y 510.051,Z 215.949,A -85,B 0,C 180,E1 -5577.631,E2 -5577.631} C_VEL
LIN {X 0,Y 510.057,Z 215.947,A -85,B 0,C 180,E1 -5580,E2 -5580} C_VEL
LIN {X 0,Y 510.052,Z 215.944,A -85,B 0,C 180,E1 -5582.369,E2 -5582.369} C_VEL
LIN {X 0,Y 509.975,Z 215.963,A -85,B 0,C 180,E1 -5585.536,E2 -5585.536} C_VEL
LIN {X 0,Y 509.904,Z 215.961,A -85,B 0,C 180,E1 -5588.721,E2 -5588.721} C_VEL
LIN {X 0,Y 509.906,Z 215.965,A -85,B 0,C 180,E1 -5591.932,E2 -5591.932} C_VEL
LIN {X 0,Y 509.896,Z 215.97,A -85,B 0,C 180,E1 -5595.242,E2 -5595.242} C_VEL
LIN {X 0,Y 509.858,Z 215.967,A -85,B 0,C 180,E1 -5598.484,E2 -5598.484} C_VEL
LIN {X 0,Y 509.848,Z 215.974,A -85,B 0,C 180,E1 -5601.002,E2 -5601.002} C_VEL
LIN {X 0,Y 509.821,Z 215.981,A -85,B 0,C 180,E1 -5603.564,E2 -5603.564} C_VEL
LIN {X 0,Y 509.879,Z 215.965,A -85,B 0,C 180,E1 -5606.371,E2 -5606.371} C_VEL
LIN {X 0,Y 509.873,Z 215.97,A -85,B 0,C 180,E1 -5608.845,E2 -5608.845} C_VEL
LIN {X 0,Y 509.821,Z 215.981,A -85,B 0,C 180,E1 -5611.59,E2 -5611.59} C_VEL
LIN {X 0,Y 509.848,Z 215.971,A -85,B 0,C 180,E1 -5614.414,E2 -5614.414} C_VEL
LIN {X 0,Y 509.809,Z 215.983,A -85,B 0,C 180,E1 -5617.342,E2 -5617.342} C_VEL
LIN {X 0,Y 509.84,Z 215.973,A -85,B 0,C 180,E1 -5620.382,E2 -5620.382} C_VEL
LIN {X 0,Y 509.807,Z 215.981,A -85,B 0,C 180,E1 -5623.06,E2 -5623.06} C_VEL
LIN {X 0,Y 509.824,Z 215.976,A -85,B 0,C 180,E1 -5625.794,E2 -5625.794} C_VEL
LIN {X 0,Y 509.854,Z 215.973,A -85,B 0,C 180,E1 -5628.574,E2 -5628.574} C_VEL
LIN {X 0,Y 509.852,Z 215.977,A -85,B 0,C 180,E1 -5631.787,E2 -5631.787} C_VEL
LIN {X 0,Y 509.822,Z 215.982,A -85,B 0,C 180,E1 -5633.709,E2 -5633.709} C_VEL
LIN {X 0,Y 509.152,Z 216.062,A -85,B 0,C 180,E1 -5634.369,E2 -5634.369} C_VEL
LIN {X 0,Y 506.342,Z 216.417,A -85,B 0,C 180,E1 -5635.441,E2 -5635.441} C_VEL
LIN {X 0,Y 503.957,Z 216.714,A -85,B 0,C 180,E1 -5636.304,E2 -5636.304} C_VEL
LIN {X 0,Y 502.91,Z 216.84,A -85,B 0,C 180,E1 -5636.97,E2 -5636.97} C_VEL
LIN {X 0,Y 502.812,Z 216.851,A -85,B 0,C 180,E1 -5637.196,E2 -5637.196} C_VEL
LIN {X 0,Y 502.818,Z 216.847,A -85,B 0,C 180,E1 -5640.065,E2 -5640.065} C_VEL
LIN {X 0,Y 502.883,Z 217.02,A -85,B 0,C 180,E1 -5643.234,E2 -5643.234} C_VEL
LIN {X 0,Y 503.67,Z 222.755,A -85,B 0,C 180,E1 -5644.37,E2 -5644.37} C_VEL
LIN {X 0,Y 503.336,Z 239.305,A -85,B 0,C 180,E1 -5647.492,E2 -5647.492} C_VEL
LIN {X 0,Y 503.272,Z 243.288,A -85,B 0,C 180,E1 -5648.235,E2 -5648.235} C_VEL
LIN {X 0,Y 505.475,Z 255.515,A -85,B 0,C 180,E1 -5648.496,E2 -5648.496} C_VEL
LIN {X 0,Y 504.855,Z 350.632,A -85,B 0,C 180,E1 -5649.873,E2 -5649.873} C_VEL
LIN {X 0,Y 504.658,Z 364.078,A -85,B 0,C 180,E1 -5650.236,E2 -5650.236} C_VEL
LIN {X 0,Y 504.353,Z 376.357,A -85,B 0,C 180,E1 -5650.726,E2 -5650.726} C_VEL
LIN {X 0,Y 504.121,Z 388.326,A -85,B 0,C 180,E1 -5651.38,E2 -5651.38} C_VEL
LIN {X 0,Y 503.743,Z 399.023,A -85,B 0,C 180,E1 -5652.125,E2 -5652.125} C_VEL
LIN {X 0,Y 503.421,Z 409.711,A -85,B 0,C 180,E1 -5653.057,E2 -5653.057} C_VEL
LIN {X 0,Y 503.06,Z 418.398,A -85,B 0,C 180,E1 -5653.983,E2 -5653.983} C_VEL
LIN {X 0,Y 502.745,Z 426.637,A -85,B 0,C 180,E1 -5655.051,E2 -5655.051} C_VEL
LIN {X 0,Y 502.511,Z 434.092,A -85,B 0,C 180,E1 -5656.246,E2 -5656.246} C_VEL
LIN {X 0,Y 502.381,Z 440.267,A -85,B 0,C 180,E1 -5657.477,E2 -5657.477} C_VEL
LIN {X 0,Y 502.256,Z 445.135,A -85,B 0,C 180,E1 -5658.703,E2 -5658.703} C_VEL
LIN {X 0,Y 502.167,Z 448.855,A -85,B 0,C 180,E1 -5659.925,E2 -5659.925} C_VEL
LIN {X 0,Y 502.068,Z 451.534,A -85,B 0,C 180,E1 -5661.142,E2 -5661.142} C_VEL
LIN {X 0,Y 502.06,Z 452.791,A -85,B 0,C 180,E1 -5661.953,E2 -5661.953} C_VEL
LIN {X 0,Y 502.112,Z 453.642,A -85,B 0,C 180,E1 -5662.763,E2 -5662.763} C_VEL
LIN {X 0,Y 502.095,Z 454.083,A -85,B 0,C 180,E1 -5664.377,E2 -5664.377} C_VEL
LIN {X 0,Y 502.094,Z 452.985,A -85,B 0,C 180,E1 -5665.987,E2 -5665.987} C_VEL
LIN {X 0,Y 502.125,Z 451.804,A -85,B 0,C 180,E1 -5666.791,E2 -5666.791} C_VEL
LIN {X 0,Y 502.133,Z 450.223,A -85,B 0,C 180,E1 -5667.593,E2 -5667.593} C_VEL
LIN {X 0,Y 502.164,Z 447.056,A -85,B 0,C 180,E1 -5668.797,E2 -5668.797} C_VEL
LIN {X 0,Y 502.181,Z 442.849,A -85,B 0,C 180,E1 -5670,E2 -5670} C_VEL
LIN {X 0,Y 502.512,Z 436.466,A -85,B 0,C 180,E1 -5671.402,E2 -5671.402} C_VEL
LIN {X 0,Y 502.61,Z 429.52,A -85,B 0,C 180,E1 -5672.605,E2 -5672.605} C_VEL
LIN {X 0,Y 502.937,Z 420.844,A -85,B 0,C 180,E1 -5673.806,E2 -5673.806} C_VEL
LIN {X 0,Y 503.253,Z 411.978,A -85,B 0,C 180,E1 -5674.806,E2 -5674.806} C_VEL
LIN {X 0,Y 503.615,Z 402.24,A -85,B 0,C 180,E1 -5675.706,E2 -5675.706} C_VEL
LIN {X 0,Y 503.979,Z 391.489,A -85,B 0,C 180,E1 -5676.506,E2 -5676.506} C_VEL
LIN {X 0,Y 504.296,Z 379.482,A -85,B 0,C 180,E1 -5677.205,E2 -5677.205} C_VEL
LIN {X 0,Y 504.632,Z 366.906,A -85,B 0,C 180,E1 -5677.754,E2 -5677.754} C_VEL
LIN {X 0,Y 504.824,Z 353.647,A -85,B 0,C 180,E1 -5678.147,E2 -5678.147} C_VEL
LIN {X 0,Y 504.989,Z 335.431,A -85,B 0,C 180,E1 -5678.45,E2 -5678.45} C_VEL
LIN {X 0,Y 505.365,Z 254.47,A -85,B 0,C 180,E1 -5679.607,E2 -5679.607} C_VEL
LIN {X 0,Y 503.263,Z 243.273,A -85,B 0,C 180,E1 -5679.85,E2 -5679.85} C_VEL
LIN {X 0,Y 503.574,Z 228.218,A -85,B 0,C 180,E1 -5682.686,E2 -5682.686} C_VEL
LIN {X 0,Y 503.57,Z 220.638,A -85,B 0,C 180,E1 -5684.137,E2 -5684.137} C_VEL
LIN {X 0,Y 502.907,Z 216.845,A -85,B 0,C 180,E1 -5684.905,E2 -5684.905} C_VEL
LIN {X 0,Y 502.832,Z 216.849,A -85,B 0,C 180,E1 -5688.116,E2 -5688.116} C_VEL
LIN {X 0,Y 502.833,Z 216.851,A -85,B 0,C 180,E1 -5690.536,E2 -5690.536} C_VEL
LIN {X 0,Y 502.794,Z 216.853,A -85,B 0,C 180,E1 -5693.04,E2 -5693.04} C_VEL
LIN {X 0,Y 502.802,Z 216.848,A -85,B 0,C 180,E1 -5695.678,E2 -5695.678} C_VEL
LIN {X 0,Y 502.799,Z 216.853,A -85,B 0,C 180,E1 -5698.375,E2 -5698.375} C_VEL
LIN {X 0,Y 502.799,Z 216.852,A -85,B 0,C 180,E1 -5701.143,E2 -5701.143} C_VEL
LIN {X 0,Y 502.806,Z 216.849,A -85,B 0,C 180,E1 -5703.994,E2 -5703.994} C_VEL
LIN {X 0,Y 502.778,Z 216.854,A -85,B 0,C 180,E1 -5707.177,E2 -5707.177} C_VEL
LIN {X 0,Y 502.79,Z 216.851,A -85,B 0,C 180,E1 -5710.015,E2 -5710.015} C_VEL
LIN {X 0,Y 502.805,Z 216.851,A -85,B 0,C 180,E1 -5712.199,E2 -5712.199} C_VEL
LIN {X 0,Y 502.787,Z 216.851,A -85,B 0,C 180,E1 -5715.47,E2 -5715.47} C_VEL
LIN {X 0,Y 502.796,Z 216.85,A -85,B 0,C 180,E1 -5717.86,E2 -5717.86} C_VEL
LIN {X 0,Y 502.802,Z 216.852,A -85,B 0,C 180,E1 -5721.024,E2 -5721.024} C_VEL
LIN {X 0,Y 502.772,Z 216.855,A -85,B 0,C 180,E1 -5724.169,E2 -5724.169} C_VEL
LIN {X 0,Y 502.834,Z 216.849,A -85,B 0,C 180,E1 -5726.993,E2 -5726.993} C_VEL
LIN {X 0,Y 502.816,Z 216.848,A -85,B 0,C 180,E1 -5730.065,E2 -5730.065} C_VEL
LIN {X 0,Y 502.824,Z 216.853,A -85,B 0,C 180,E1 -5732.532,E2 -5732.532} C_VEL
LIN {X 0,Y 502.774,Z 216.853,A -85,B 0,C 180,E1 -5735.312,E2 -5735.312} C_VEL
LIN {X 0,Y 502.781,Z 216.851,A -85,B 0,C 180,E1 -5737.826,E2 -5737.826} C_VEL
LIN {X 0,Y 502.822,Z 216.852,A -85,B 0,C 180,E1 -5740.4,E2 -5740.4} C_VEL
LIN {X 0,Y 502.813,Z 216.852,A -85,B 0,C 180,E1 -5742.931,E2 -5742.931} C_VEL
LIN {X 0,Y 502.834,Z 216.845,A -85,B 0,C 180,E1 -5745.429,E2 -5745.429} C_VEL
LIN {X 0,Y 502.877,Z 216.847,A -85,B 0,C 180,E1 -5748.717,E2 -5748.717} C_VEL
LIN {X 0,Y 502.881,Z 216.84,A -85,B 0,C 180,E1 -5751.966,E2 -5751.966} C_VEL
LIN {X 0,Y 502.929,Z 216.838,A -85,B 0,C 180,E1 -5754.386,E2 -5754.386} C_VEL
LIN {X 0,Y 503.024,Z 216.821,A -85,B 0,C 180,E1 -5757.598,E2 -5757.598} C_VEL
LIN {X 0,Y 503.033,Z 216.826,A -85,B 0,C 180,E1 -5760.8,E2 -5760.8} C_VEL
LIN {X 0,Y 502.873,Z 216.841,A -85,B 0,C 180,E1 -5763.205,E2 -5763.205} C_VEL
LIN {X 0,Y 502.927,Z 216.839,A -85,B 0,C 180,E1 -5766.419,E2 -5766.419} C_VEL
LIN {X 0,Y 502.869,Z 216.845,A -85,B 0,C 180,E1 -5768.843,E2 -5768.843} C_VEL
LIN {X 0,Y 502.846,Z 216.845,A -85,B 0,C 180,E1 -5772.102,E2 -5772.102} C_VEL
LIN {X 0,Y 502.849,Z 216.843,A -85,B 0,C 180,E1 -5775.4,E2 -5775.4} C_VEL
LIN {X 0,Y 502.826,Z 216.852,A -85,B 0,C 180,E1 -5778.752,E2 -5778.752} C_VEL
LIN {X 0,Y 502.784,Z 216.851,A -85,B 0,C 180,E1 -5781.311,E2 -5781.311} C_VEL
LIN {X 0,Y 502.782,Z 216.852,A -85,B 0,C 180,E1 -5783.914,E2 -5783.914} C_VEL
LIN {X 0,Y 502.835,Z 216.854,A -85,B 0,C 180,E1 -5786.568,E2 -5786.568} C_VEL
LIN {X 0,Y 502.815,Z 216.848,A -85,B 0,C 180,E1 -5789.935,E2 -5789.935} C_VEL
LIN {X 0,Y 502.83,Z 216.848,A -85,B 0,C 180,E1 -5793.032,E2 -5793.032} C_VEL
LIN {X 0,Y 502.772,Z 216.854,A -85,B 0,C 180,E1 -5795.951,E2 -5795.951} C_VEL
LIN {X 0,Y 502.797,Z 216.852,A -85,B 0,C 180,E1 -5798.977,E2 -5798.977} C_VEL
LIN {X 0,Y 502.804,Z 216.852,A -85,B 0,C 180,E1 -5802.199,E2 -5802.199} C_VEL
LIN {X 0,Y 502.786,Z 216.85,A -85,B 0,C 180,E1 -5805.47,E2 -5805.47} C_VEL
LIN {X 0,Y 502.795,Z 216.85,A -85,B 0,C 180,E1 -5807.861,E2 -5807.861} C_VEL
LIN {X 0,Y 502.801,Z 216.851,A -85,B 0,C 180,E1 -5811.024,E2 -5811.024} C_VEL
LIN {X 0,Y 502.772,Z 216.856,A -85,B 0,C 180,E1 -5814.17,E2 -5814.17} C_VEL
LIN {X 0,Y 502.834,Z 216.847,A -85,B 0,C 180,E1 -5816.994,E2 -5816.994} C_VEL
LIN {X 0,Y 502.816,Z 216.849,A -85,B 0,C 180,E1 -5820.065,E2 -5820.065} C_VEL
LIN {X 0,Y 502.824,Z 216.855,A -85,B 0,C 180,E1 -5822.533,E2 -5822.533} C_VEL
LIN {X 0,Y 502.814,Z 216.993,A -85,B 0,C 180,E1 -5825.44,E2 -5825.44} C_VEL
LIN {X 0,Y 504.428,Z 226.002,A -85,B 0,C 180,E1 -5827.039,E2 -5827.039} C_VEL
LIN {X 0,Y 503.976,Z 242.648,A -85,B 0,C 180,E1 -5829.81,E2 -5829.81} C_VEL
LIN {X 0,Y 503.468,Z 260.504,A -85,B 0,C 180,E1 -5832.745,E2 -5832.745} C_VEL
LIN {X 0,Y 503.26,Z 269.405,A -85,B 0,C 180,E1 -5834.197,E2 -5834.197} C_VEL
LIN {X 0,Y 505.33,Z 283.364,A -85,B 0,C 180,E1 -5834.464,E2 -5834.464} C_VEL
LIN {X 0,Y 504.859,Z 377.449,A -85,B 0,C 180,E1 -5835.823,E2 -5835.823} C_VEL
LIN {X 0,Y 504.551,Z 390.766,A -85,B 0,C 180,E1 -5836.174,E2 -5836.174} C_VEL
LIN {X 0,Y 504.239,Z 402.952,A -85,B 0,C 180,E1 -5836.653,E2 -5836.653} C_VEL
LIN {X 0,Y 503.908,Z 415.048,A -85,B 0,C 180,E1 -5837.298,E2 -5837.298} C_VEL
LIN {X 0,Y 503.606,Z 425.56,A -85,B 0,C 180,E1 -5838.019,E2 -5838.019} C_VEL
LIN {X 0,Y 503.263,Z 436.234,A -85,B 0,C 180,E1 -5838.93,E2 -5838.93} C_VEL
LIN {X 0,Y 502.893,Z 445.851,A -85,B 0,C 180,E1 -5839.939,E2 -5839.939} C_VEL
LIN {X 0,Y 502.638,Z 453.735,A -85,B 0,C 180,E1 -5840.95,E2 -5840.95} C_VEL
LIN {X 0,Y 502.4,Z 461.435,A -85,B 0,C 180,E1 -5842.161,E2 -5842.161} C_VEL
LIN {X 0,Y 502.235,Z 468.532,A -85,B 0,C 180,E1 -5843.572,E2 -5843.572} C_VEL
LIN {X 0,Y 502.174,Z 473.255,A -85,B 0,C 180,E1 -5844.781,E2 -5844.781} C_VEL
LIN {X 0,Y 502.138,Z 476.862,A -85,B 0,C 180,E1 -5845.987,E2 -5845.987} C_VEL
LIN {X 0,Y 502.12,Z 478.723,A -85,B 0,C 180,E1 -5846.791,E2 -5846.791} C_VEL
LIN {X 0,Y 502.091,Z 480.117,A -85,B 0,C 180,E1 -5847.593,E2 -5847.593} C_VEL
LIN {X 0,Y 501.991,Z 481.717,A -85,B 0,C 180,E1 -5849.198,E2 -5849.198} C_VEL
LIN {X 0,Y 501.982,Z 481.932,A -85,B 0,C 180,E1 -5850,E2 -5850} C_VEL
LIN {X 0,Y 502.036,Z 481.109,A -85,B 0,C 180,E1 -5851.604,E2 -5851.604} C_VEL
LIN {X 0,Y 502.091,Z 480.115,A -85,B 0,C 180,E1 -5852.407,E2 -5852.407} C_VEL
LIN {X 0,Y 502.12,Z 478.719,A -85,B 0,C 180,E1 -5853.21,E2 -5853.21} C_VEL
LIN {X 0,Y 502.101,Z 475.781,A -85,B 0,C 180,E1 -5854.415,E2 -5854.415} C_VEL
LIN {X 0,Y 502.207,Z 471.808,A -85,B 0,C 180,E1 -5855.622,E2 -5855.622} C_VEL
LIN {X 0,Y 502.33,Z 465.798,A -85,B 0,C 180,E1 -5857.012,E2 -5857.012} C_VEL
LIN {X 0,Y 502.478,Z 459.017,A -85,B 0,C 180,E1 -5858.243,E2 -5858.243} C_VEL
LIN {X 0,Y 502.717,Z 450.73,A -85,B 0,C 180,E1 -5859.455,E2 -5859.455} C_VEL
LIN {X 0,Y 502.993,Z 442.236,A -85,B 0,C 180,E1 -5860.465,E2 -5860.465} C_VEL
LIN {X 0,Y 503.417,Z 431.744,A -85,B 0,C 180,E1 -5861.475,E2 -5861.475} C_VEL
LIN {X 0,Y 503.701,Z 420.223,A -85,B 0,C 180,E1 -5862.367,E2 -5862.367} C_VEL
LIN {X 0,Y 504.137,Z 408.054,A -85,B 0,C 180,E1 -5863.093,E2 -5863.093} C_VEL
LIN {X 0,Y 504.44,Z 395.703,A -85,B 0,C 180,E1 -5863.649,E2 -5863.649} C_VEL
LIN {X 0,Y 504.735,Z 383.029,A -85,B 0,C 180,E1 -5864.052,E2 -5864.052} C_VEL
LIN {X 0,Y 504.902,Z 369.782,A -85,B 0,C 180,E1 -5864.304,E2 -5864.304} C_VEL
LIN {X 0,Y 505.262,Z 282.201,A -85,B 0,C 180,E1 -5865.557,E2 -5865.557} C_VEL
LIN {X 0,Y 503.224,Z 269.284,A -85,B 0,C 180,E1 -5865.821,E2 -5865.821} C_VEL
LIN {X 0,Y 503.744,Z 250.363,A -85,B 0,C 180,E1 -5868.928,E2 -5868.928} C_VEL
LIN {X 0,Y 504.256,Z 233.876,A -85,B 0,C 180,E1 -5871.675,E2 -5871.675} C_VEL
LIN {X 0,Y 504.412,Z 225.26,A -85,B 0,C 180,E1 -5873.135,E2 -5873.135} C_VEL
LIN {X 0,Y 502.775,Z 216.859,A -85,B 0,C 180,E1 -5874.687,E2 -5874.687} C_VEL
LIN {X 0,Y 502.804,Z 216.859,A -85,B 0,C 180,E1 -5877.469,E2 -5877.469} C_VEL
LIN {X 0,Y 502.81,Z 216.85,A -85,B 0,C 180,E1 -5880.211,E2 -5880.211} C_VEL
LIN {X 0,Y 502.833,Z 216.849,A -85,B 0,C 180,E1 -5883.031,E2 -5883.031} C_VEL
LIN {X 0,Y 502.769,Z 216.856,A -85,B 0,C 180,E1 -5885.952,E2 -5885.952} C_VEL
LIN {X 0,Y 502.802,Z 216.852,A -85,B 0,C 180,E1 -5888.976,E2 -5888.976} C_VEL
LIN {X 0,Y 502.804,Z 216.85,A -85,B 0,C 180,E1 -5892.199,E2 -5892.199} C_VEL
LIN {X 0,Y 502.787,Z 216.86,A -85,B 0,C 180,E1 -5895.47,E2 -5895.47} C_VEL
LIN {X 0,Y 502.796,Z 216.854,A -85,B 0,C 180,E1 -5897.86,E2 -5897.86} C_VEL
LIN {X 0,Y 502.797,Z 216.852,A -85,B 0,C 180,E1 -5901.023,E2 -5901.023} C_VEL
LIN {X 0,Y 502.771,Z 216.853,A -85,B 0,C 180,E1 -5904.17,E2 -5904.17} C_VEL
LIN {X 0,Y 502.831,Z 216.846,A -85,B 0,C 180,E1 -5906.994,E2 -5906.994} C_VEL
LIN {X 0,Y 502.816,Z 216.846,A -85,B 0,C 180,E1 -5910.065,E2 -5910.065} C_VEL
LIN {X 0,Y 502.845,Z 216.85,A -85,B 0,C 180,E1 -5913.444,E2 -5913.444} C_VEL
LIN {X 0,Y 502.775,Z 216.854,A -85,B 0,C 180,E1 -5916.085,E2 -5916.085} C_VEL
LIN {X 0,Y 502.784,Z 216.85,A -85,B 0,C 180,E1 -5918.689,E2 -5918.689} C_VEL
LIN {X 0,Y 502.827,Z 216.852,A -85,B 0,C 180,E1 -5921.248,E2 -5921.248} C_VEL
LIN {X 0,Y 502.85,Z 216.842,A -85,B 0,C 180,E1 -5924.6,E2 -5924.6} C_VEL
LIN {X 0,Y 502.878,Z 216.838,A -85,B 0,C 180,E1 -5928.039,E2 -5928.039} C_VEL
LIN {X 0,Y 502.869,Z 216.845,A -85,B 0,C 180,E1 -5931.157,E2 -5931.157} C_VEL
LIN {X 0,Y 502.928,Z 216.839,A -85,B 0,C 180,E1 -5933.581,E2 -5933.581} C_VEL
LIN {X 0,Y 502.864,Z 216.842,A -85,B 0,C 180,E1 -5936.795,E2 -5936.795} C_VEL
LIN {X 0,Y 502.897,Z 216.834,A -85,B 0,C 180,E1 -5938.398,E2 -5938.398} C_VEL
LIN {X 0,Y 503.011,Z 216.824,A -85,B 0,C 180,E1 -5940.801,E2 -5940.801} C_VEL
LIN {X 0,Y 503.02,Z 216.819,A -85,B 0,C 180,E1 -5942.402,E2 -5942.402} C_VEL
LIN {X 0,Y 502.929,Z 216.839,A -85,B 0,C 180,E1 -5945.614,E2 -5945.614} C_VEL
LIN {X 0,Y 502.864,Z 216.839,A -85,B 0,C 180,E1 -5948.844,E2 -5948.844} C_VEL
LIN {X 0,Y 502.846,Z 216.843,A -85,B 0,C 180,E1 -5952.102,E2 -5952.102} C_VEL
LIN {X 0,Y 502.85,Z 216.851,A -85,B 0,C 180,E1 -5955.4,E2 -5955.4} C_VEL
LIN {X 0,Y 502.824,Z 216.844,A -85,B 0,C 180,E1 -5958.752,E2 -5958.752} C_VEL
LIN {X 0,Y 502.782,Z 216.858,A -85,B 0,C 180,E1 -5961.311,E2 -5961.311} C_VEL
LIN {X 0,Y 502.77,Z 216.855,A -85,B 0,C 180,E1 -5963.915,E2 -5963.915} C_VEL
LIN {X 0,Y 502.837,Z 216.842,A -85,B 0,C 180,E1 -5966.568,E2 -5966.568} C_VEL
LIN {X 0,Y 502.823,Z 216.854,A -85,B 0,C 180,E1 -5969.288,E2 -5969.288} C_VEL
LIN {X 0,Y 502.785,Z 216.852,A -85,B 0,C 180,E1 -5972.085,E2 -5972.085} C_VEL
LIN {X 0,Y 502.799,Z 216.852,A -85,B 0,C 180,E1 -5974.966,E2 -5974.966} C_VEL
LIN {X 0,Y 502.795,Z 216.85,A -85,B 0,C 180,E1 -5978.486,E2 -5978.486} C_VEL
LIN {X 0,Y 502.802,Z 216.854,A -85,B 0,C 180,E1 -5981.068,E2 -5981.068} C_VEL
LIN {X 0,Y 502.781,Z 216.853,A -85,B 0,C 180,E1 -5984.34,E2 -5984.34} C_VEL
LIN {X 0,Y 502.756,Z 216.854,A -85,B 0,C 180,E1 -5986.767,E2 -5986.767} C_VEL
LIN {X 0,Y 502.801,Z 216.855,A -85,B 0,C 180,E1 -5989.008,E2 -5989.008} C_VEL
LIN {X 0,Y 502.794,Z 216.854,A -85,B 0,C 180,E1 -5992.046,E2 -5992.046} C_VEL
LIN {X 0,Y 502.797,Z 216.856,A -85,B 0,C 180,E1 -5995.034,E2 -5995.034} C_VEL
LIN {X 0,Y 502.812,Z 216.851,A -85,B 0,C 180,E1 -5997.196,E2 -5997.196} C_VEL
LIN {X 0,Y 502.11,Z 216.939,A -85,B 0,C 180,E1 -5997.864,E2 -5997.864} C_VEL
LIN {X 0,Y 499.249,Z 217.295,A -85,B 0,C 180,E1 -5998.95,E2 -5998.95} C_VEL
LIN {X 0,Y 496.852,Z 217.592,A -85,B 0,C 180,E1 -5999.825,E2 -5999.825} C_VEL
LIN {X 0,Y 495.824,Z 217.717,A -85,B 0,C 180,E1 -6000.501,E2 -6000.501} C_VEL
LIN {X 0,Y 495.74,Z 217.728,A -85,B 0,C 180,E1 -6000.729,E2 -6000.729} C_VEL
LIN {X 0,Y 495.834,Z 217.928,A -85,B 0,C 180,E1 -6003.073,E2 -6003.073} C_VEL
LIN {X 0,Y 496.704,Z 223.562,A -85,B 0,C 180,E1 -6004.209,E2 -6004.209} C_VEL
LIN {X 0,Y 496.39,Z 239.436,A -85,B 0,C 180,E1 -6007.238,E2 -6007.238} C_VEL
LIN {X 0,Y 496.332,Z 243.695,A -85,B 0,C 180,E1 -6008.01,E2 -6008.01} C_VEL
LIN {X 0,Y 498.695,Z 256.282,A -85,B 0,C 180,E1 -6008.279,E2 -6008.279} C_VEL
LIN {X 0,Y 498.011,Z 350.742,A -85,B 0,C 180,E1 -6009.665,E2 -6009.665} C_VEL
LIN {X 0,Y 497.805,Z 364.201,A -85,B 0,C 180,E1 -6010.033,E2 -6010.033} C_VEL
LIN {X 0,Y 497.448,Z 377.051,A -85,B 0,C 180,E1 -6010.555,E2 -6010.555} C_VEL
LIN {X 0,Y 497.212,Z 387.959,A -85,B 0,C 180,E1 -6011.159,E2 -6011.159} C_VEL
LIN {X 0,Y 496.782,Z 399.483,A -85,B 0,C 180,E1 -6011.973,E2 -6011.973} C_VEL
LIN {X 0,Y 496.44,Z 410.119,A -85,B 0,C 180,E1 -6012.917,E2 -6012.917} C_VEL
LIN {X 0,Y 496.047,Z 419.626,A -85,B 0,C 180,E1 -6013.962,E2 -6013.962} C_VEL
LIN {X 0,Y 495.686,Z 428.755,A -85,B 0,C 180,E1 -6015.214,E2 -6015.214} C_VEL
LIN {X 0,Y 495.43,Z 436.079,A -85,B 0,C 180,E1 -6016.464,E2 -6016.464} C_VEL
LIN {X 0,Y 495.304,Z 441.895,A -85,B 0,C 180,E1 -6017.711,E2 -6017.711} C_VEL
LIN {X 0,Y 495.139,Z 446.441,A -85,B 0,C 180,E1 -6018.953,E2 -6018.953} C_VEL
LIN {X 0,Y 495.029,Z 449.879,A -85,B 0,C 180,E1 -6020.191,E2 -6020.191} C_VEL
LIN {X 0,Y 494.983,Z 451.579,A -85,B 0,C 180,E1 -6021.015,E2 -6021.015} C_VEL
LIN {X 0,Y 495.004,Z 453.764,A -85,B 0,C 180,E1 -6022.659,E2 -6022.659} C_VEL
LIN {X 0,Y 495,Z 454.269,A -85,B 0,C 180,E1 -6023.649,E2 -6023.649} C_VEL
LIN {X 0,Y 494.971,Z 453.975,A -85,B 0,C 180,E1 -6025.113,E2 -6025.113} C_VEL
LIN {X 0,Y 494.992,Z 453.272,A -85,B 0,C 180,E1 -6025.929,E2 -6025.929} C_VEL
LIN {X 0,Y 495.043,Z 452.15,A -85,B 0,C 180,E1 -6026.745,E2 -6026.745} C_VEL
LIN {X 0,Y 495.065,Z 450.603,A -85,B 0,C 180,E1 -6027.559,E2 -6027.559} C_VEL
LIN {X 0,Y 495.067,Z 447.51,A -85,B 0,C 180,E1 -6028.78,E2 -6028.78} C_VEL
LIN {X 0,Y 495.099,Z 443.378,A -85,B 0,C 180,E1 -6030,E2 -6030} C_VEL
LIN {X 0,Y 495.441,Z 437.076,A -85,B 0,C 180,E1 -6031.422,E2 -6031.422} C_VEL
LIN {X 0,Y 495.555,Z 430.252,A -85,B 0,C 180,E1 -6032.642,E2 -6032.642} C_VEL
LIN {X 0,Y 495.897,Z 421.701,A -85,B 0,C 180,E1 -6033.86,E2 -6033.86} C_VEL
LIN {X 0,Y 496.233,Z 412.957,A -85,B 0,C 180,E1 -6034.875,E2 -6034.875} C_VEL
LIN {X 0,Y 496.674,Z 402.203,A -85,B 0,C 180,E1 -6035.888,E2 -6035.888} C_VEL
LIN {X 0,Y 497.064,Z 391.365,A -85,B 0,C 180,E1 -6036.699,E2 -6036.699} C_VEL
LIN {X 0,Y 497.398,Z 379.267,A -85,B 0,C 180,E1 -6037.408,E2 -6037.408} C_VEL
LIN {X 0,Y 497.745,Z 366.531,A -85,B 0,C 180,E1 -6037.964,E2 -6037.964} C_VEL
LIN {X 0,Y 497.957,Z 353.333,A -85,B 0,C 180,E1 -6038.352,E2 -6038.352} C_VEL
LIN {X 0,Y 498.139,Z 334.678,A -85,B 0,C 180,E1 -6038.66,E2 -6038.66} C_VEL
LIN {X 0,Y 498.552,Z 255.479,A -85,B 0,C 180,E1 -6039.805,E2 -6039.805} C_VEL
LIN {X 0,Y 496.316,Z 243.439,A -85,B 0,C 180,E1 -6040.067,E2 -6040.067} C_VEL
LIN {X 0,Y 496.62,Z 228.75,A -85,B 0,C 180,E1 -6042.858,E2 -6042.858} C_VEL
LIN {X 0,Y 496.627,Z 222.162,A -85,B 0,C 180,E1 -6044.129,E2 -6044.129} C_VEL
LIN {X 0,Y 495.848,Z 217.724,A -85,B 0,C 180,E1 -6045.027,E2 -6045.027} C_VEL
LIN {X 0,Y 495.782,Z 217.729,A -85,B 0,C 180,E1 -6048.237,E2 -6048.237} C_VEL
LIN {X 0,Y 495.778,Z 217.732,A -85,B 0,C 180,E1 -6050.756,E2 -6050.756} C_VEL
LIN {X 0,Y 495.75,Z 217.728,A -85,B 0,C 180,E1 -6053.387,E2 -6053.387} C_VEL
LIN {X 0,Y 495.762,Z 217.727,A -85,B 0,C 180,E1 -6056.069,E2 -6056.069} C_VEL
LIN {X 0,Y 495.747,Z 217.734,A -85,B 0,C 180,E1 -6058.816,E2 -6058.816} C_VEL
LIN {X 0,Y 495.758,Z 217.726,A -85,B 0,C 180,E1 -6061.725,E2 -6061.725} C_VEL
LIN {X 0,Y 495.77,Z 217.733,A -85,B 0,C 180,E1 -6064.694,E2 -6064.694} C_VEL
LIN {X 0,Y 495.73,Z 217.73,A -85,B 0,C 180,E1 -6067.562,E2 -6067.562} C_VEL
LIN {X 0,Y 495.768,Z 217.734,A -85,B 0,C 180,E1 -6070.7,E2 -6070.7} C_VEL
LIN {X 0,Y 495.73,Z 217.731,A -85,B 0,C 180,E1 -6074.001,E2 -6074.001} C_VEL
LIN {X 0,Y 495.719,Z 217.734,A -85,B 0,C 180,E1 -6077.116,E2 -6077.116} C_VEL
LIN {X 0,Y 495.76,Z 217.727,A -85,B 0,C 180,E1 -6079.953,E2 -6079.953} C_VEL
LIN {X 0,Y 495.72,Z 217.738,A -85,B 0,C 180,E1 -6082.554,E2 -6082.554} C_VEL
LIN {X 0,Y 495.778,Z 217.724,A -85,B 0,C 180,E1 -6085.457,E2 -6085.457} C_VEL
LIN {X 0,Y 495.757,Z 217.731,A -85,B 0,C 180,E1 -6088.364,E2 -6088.364} C_VEL
LIN {X 0,Y 495.786,Z 217.723,A -85,B 0,C 180,E1 -6091.507,E2 -6091.507} C_VEL
LIN {X 0,Y 495.755,Z 217.727,A -85,B 0,C 180,E1 -6093.93,E2 -6093.93} C_VEL
LIN {X 0,Y 495.76,Z 217.728,A -85,B 0,C 180,E1 -6097.14,E2 -6097.14} C_VEL
LIN {X 0,Y 495.77,Z 217.727,A -85,B 0,C 180,E1 -6100.109,E2 -6100.109} C_VEL
LIN {X 0,Y 495.76,Z 217.734,A -85,B 0,C 180,E1 -6102.68,E2 -6102.68} C_VEL
LIN {X 0,Y 495.783,Z 217.724,A -85,B 0,C 180,E1 -6105.217,E2 -6105.217} C_VEL
LIN {X 0,Y 495.852,Z 217.722,A -85,B 0,C 180,E1 -6108.555,E2 -6108.555} C_VEL
LIN {X 0,Y 495.837,Z 217.717,A -85,B 0,C 180,E1 -6111.851,E2 -6111.851} C_VEL
LIN {X 0,Y 495.884,Z 217.715,A -85,B 0,C 180,E1 -6114.306,E2 -6114.306} C_VEL
LIN {X 0,Y 495.993,Z 217.697,A -85,B 0,C 180,E1 -6117.564,E2 -6117.564} C_VEL
LIN {X 0,Y 495.983,Z 217.704,A -85,B 0,C 180,E1 -6120.812,E2 -6120.812} C_VEL
LIN {X 0,Y 495.989,Z 217.704,A -85,B 0,C 180,E1 -6122.436,E2 -6122.436} C_VEL
LIN {X 0,Y 495.894,Z 217.709,A -85,B 0,C 180,E1 -6125.693,E2 -6125.693} C_VEL
LIN {X 0,Y 495.873,Z 217.715,A -85,B 0,C 180,E1 -6128.148,E2 -6128.148} C_VEL
LIN {X 0,Y 495.852,Z 217.714,A -85,B 0,C 180,E1 -6131.445,E2 -6131.445} C_VEL
LIN {X 0,Y 495.795,Z 217.727,A -85,B 0,C 180,E1 -6134.783,E2 -6134.783} C_VEL
LIN {X 0,Y 495.763,Z 217.726,A -85,B 0,C 180,E1 -6137.319,E2 -6137.319} C_VEL
LIN {X 0,Y 495.771,Z 217.725,A -85,B 0,C 180,E1 -6139.89,E2 -6139.89} C_VEL
LIN {X 0,Y 495.76,Z 217.73,A -85,B 0,C 180,E1 -6142.861,E2 -6142.861} C_VEL
LIN {X 0,Y 495.76,Z 217.728,A -85,B 0,C 180,E1 -6146.07,E2 -6146.07} C_VEL
LIN {X 0,Y 495.745,Z 217.733,A -85,B 0,C 180,E1 -6148.817,E2 -6148.817} C_VEL
LIN {X 0,Y 495.755,Z 217.727,A -85,B 0,C 180,E1 -6151.725,E2 -6151.725} C_VEL
LIN {X 0,Y 495.762,Z 217.733,A -85,B 0,C 180,E1 -6154.693,E2 -6154.693} C_VEL
LIN {X 0,Y 495.721,Z 217.731,A -85,B 0,C 180,E1 -6157.562,E2 -6157.562} C_VEL
LIN {X 0,Y 495.756,Z 217.728,A -85,B 0,C 180,E1 -6160.047,E2 -6160.047} C_VEL
LIN {X 0,Y 495.715,Z 217.735,A -85,B 0,C 180,E1 -6162.884,E2 -6162.884} C_VEL
LIN {X 0,Y 495.725,Z 217.732,A -85,B 0,C 180,E1 -6165.998,E2 -6165.998} C_VEL
LIN {X 0,Y 495.741,Z 217.735,A -85,B 0,C 180,E1 -6168.709,E2 -6168.709} C_VEL
LIN {X 0,Y 495.75,Z 217.727,A -85,B 0,C 180,E1 -6171.408,E2 -6171.408} C_VEL
LIN {X 0,Y 495.746,Z 217.735,A -85,B 0,C 180,E1 -6174.462,E2 -6174.462} C_VEL
LIN {X 0,Y 495.769,Z 217.725,A -85,B 0,C 180,E1 -6177.406,E2 -6177.406} C_VEL
LIN {X 0,Y 495.767,Z 217.73,A -85,B 0,C 180,E1 -6180.254,E2 -6180.254} C_VEL
LIN {X 0,Y 495.807,Z 217.724,A -85,B 0,C 180,E1 -6183.255,E2 -6183.255} C_VEL
LIN {X 0,Y 495.764,Z 217.808,A -85,B 0,C 180,E1 -6185.264,E2 -6185.264} C_VEL
LIN {X 0,Y 497.451,Z 226.564,A -85,B 0,C 180,E1 -6186.846,E2 -6186.846} C_VEL
LIN {X 0,Y 497.108,Z 239.493,A -85,B 0,C 180,E1 -6189.032,E2 -6189.032} C_VEL
LIN {X 0,Y 496.554,Z 257.696,A -85,B 0,C 180,E1 -6192.071,E2 -6192.071} C_VEL
LIN {X 0,Y 496.245,Z 269.205,A -85,B 0,C 180,E1 -6193.975,E2 -6193.975} C_VEL
LIN {X 0,Y 498.477,Z 284.111,A -85,B 0,C 180,E1 -6194.264,E2 -6194.264} C_VEL
LIN {X 0,Y 497.974,Z 377.06,A -85,B 0,C 180,E1 -6195.623,E2 -6195.623} C_VEL
LIN {X 0,Y 497.671,Z 390.456,A -85,B 0,C 180,E1 -6195.979,E2 -6195.979} C_VEL
LIN {X 0,Y 497.322,Z 402.684,A -85,B 0,C 180,E1 -6196.464,E2 -6196.464} C_VEL
LIN {X 0,Y 496.959,Z 415.106,A -85,B 0,C 180,E1 -6197.136,E2 -6197.136} C_VEL
LIN {X 0,Y 496.614,Z 425.343,A -85,B 0,C 180,E1 -6197.848,E2 -6197.848} C_VEL
LIN {X 0,Y 496.264,Z 436.026,A -85,B 0,C 180,E1 -6198.771,E2 -6198.771} C_VEL
LIN {X 0,Y 495.854,Z 445.647,A -85,B 0,C 180,E1 -6199.795,E2 -6199.795} C_VEL
LIN {X 0,Y 495.599,Z 453.536,A -85,B 0,C 180,E1 -6200.82,E2 -6200.82} C_VEL
LIN {X 0,Y 495.343,Z 461.238,A -85,B 0,C 180,E1 -6202.049,E2 -6202.049} C_VEL
LIN {X 0,Y 495.164,Z 468.336,A -85,B 0,C 180,E1 -6203.48,E2 -6203.48} C_VEL
LIN {X 0,Y 495.106,Z 473.059,A -85,B 0,C 180,E1 -6204.706,E2 -6204.706} C_VEL
LIN {X 0,Y 495.031,Z 476.666,A -85,B 0,C 180,E1 -6205.929,E2 -6205.929} C_VEL
LIN {X 0,Y 495.041,Z 478.527,A -85,B 0,C 180,E1 -6206.745,E2 -6206.745} C_VEL
LIN {X 0,Y 494.998,Z 479.921,A -85,B 0,C 180,E1 -6207.559,E2 -6207.559} C_VEL
LIN {X 0,Y 494.962,Z 480.915,A -85,B 0,C 180,E1 -6208.373,E2 -6208.373} C_VEL
LIN {X 0,Y 494.9,Z 481.736,A -85,B 0,C 180,E1 -6210,E2 -6210} C_VEL
LIN {X 0,Y 494.962,Z 480.913,A -85,B 0,C 180,E1 -6211.627,E2 -6211.627} C_VEL
LIN {X 0,Y 494.998,Z 479.917,A -85,B 0,C 180,E1 -6212.441,E2 -6212.441} C_VEL
LIN {X 0,Y 495.042,Z 478.522,A -85,B 0,C 180,E1 -6213.255,E2 -6213.255} C_VEL
LIN {X 0,Y 495.007,Z 475.583,A -85,B 0,C 180,E1 -6214.479,E2 -6214.479} C_VEL
LIN {X 0,Y 495.124,Z 471.61,A -85,B 0,C 180,E1 -6215.702,E2 -6215.702} C_VEL
LIN {X 0,Y 495.255,Z 465.497,A -85,B 0,C 180,E1 -6217.133,E2 -6217.133} C_VEL
LIN {X 0,Y 495.426,Z 458.817,A -85,B 0,C 180,E1 -6218.361,E2 -6218.361} C_VEL
LIN {X 0,Y 495.695,Z 450.534,A -85,B 0,C 180,E1 -6219.59,E2 -6219.59} C_VEL
LIN {X 0,Y 495.988,Z 442.044,A -85,B 0,C 180,E1 -6220.615,E2 -6220.615} C_VEL
LIN {X 0,Y 496.453,Z 431.561,A -85,B 0,C 180,E1 -6221.638,E2 -6221.638} C_VEL
LIN {X 0,Y 496.752,Z 420.322,A -85,B 0,C 180,E1 -6222.523,E2 -6222.523} C_VEL
LIN {X 0,Y 497.196,Z 407.923,A -85,B 0,C 180,E1 -6223.279,E2 -6223.279} C_VEL
LIN {X 0,Y 497.556,Z 395.607,A -85,B 0,C 180,E1 -6223.842,E2 -6223.842} C_VEL
LIN {X 0,Y 497.86,Z 382.988,A -85,B 0,C 180,E1 -6224.25,E2 -6224.25} C_VEL
LIN {X 0,Y 498.04,Z 369.919,A -85,B 0,C 180,E1 -6224.506,E2 -6224.506} C_VEL
LIN {X 0,Y 498.48,Z 283.178,A -85,B 0,C 180,E1 -6225.764,E2 -6225.764} C_VEL
LIN {X 0,Y 496.254,Z 268.992,A -85,B 0,C 180,E1 -6226.073,E2 -6226.073} C_VEL
LIN {X 0,Y 496.794,Z 250.242,A -85,B 0,C 180,E1 -6229.203,E2 -6229.203} C_VEL
LIN {X 0,Y 497.324,Z 235.042,A -85,B 0,C 180,E1 -6231.775,E2 -6231.775} C_VEL
LIN {X 0,Y 497.521,Z 226.938,A -85,B 0,C 180,E1 -6233.167,E2 -6233.167} C_VEL
LIN {X 0,Y 495.729,Z 217.738,A -85,B 0,C 180,E1 -6234.889,E2 -6234.889} C_VEL
LIN {X 0,Y 495.744,Z 217.736,A -85,B 0,C 180,E1 -6237.894,E2 -6237.894} C_VEL
LIN {X 0,Y 495.752,Z 217.729,A -85,B 0,C 180,E1 -6240.687,E2 -6240.687} C_VEL
LIN {X 0,Y 495.76,Z 217.734,A -85,B 0,C 180,E1 -6243.564,E2 -6243.564} C_VEL
LIN {X 0,Y 495.717,Z 217.732,A -85,B 0,C 180,E1 -6246.545,E2 -6246.545} C_VEL
LIN {X 0,Y 495.757,Z 217.734,A -85,B 0,C 180,E1 -6249.638,E2 -6249.638} C_VEL
LIN {X 0,Y 495.736,Z 217.73,A -85,B 0,C 180,E1 -6252.506,E2 -6252.506} C_VEL
LIN {X 0,Y 495.738,Z 217.734,A -85,B 0,C 180,E1 -6255.141,E2 -6255.141} C_VEL
LIN {X 0,Y 495.751,Z 217.728,A -85,B 0,C 180,E1 -6258.218,E2 -6258.218} C_VEL
LIN {X 0,Y 495.748,Z 217.736,A -85,B 0,C 180,E1 -6261.408,E2 -6261.408} C_VEL
LIN {X 0,Y 495.744,Z 217.728,A -85,B 0,C 180,E1 -6264.462,E2 -6264.462} C_VEL
LIN {X 0,Y 495.767,Z 217.73,A -85,B 0,C 180,E1 -6267.406,E2 -6267.406} C_VEL
LIN {X 0,Y 495.764,Z 217.723,A -85,B 0,C 180,E1 -6270.253,E2 -6270.253} C_VEL
LIN {X 0,Y 495.775,Z 217.731,A -85,B 0,C 180,E1 -6273.262,E2 -6273.262} C_VEL
LIN {X 0,Y 495.743,Z 217.729,A -85,B 0,C 180,E1 -6276.612,E2 -6276.612} C_VEL
LIN {X 0,Y 495.78,Z 217.728,A -85,B 0,C 180,E1 -6279.324,E2 -6279.324} C_VEL
LIN {X 0,Y 495.782,Z 217.726,A -85,B 0,C 180,E1 -6281.828,E2 -6281.828} C_VEL
LIN {X 0,Y 495.825,Z 217.717,A -85,B 0,C 180,E1 -6284.548,E2 -6284.548} C_VEL
LIN {X 0,Y 495.83,Z 217.716,A -85,B 0,C 180,E1 -6287.965,E2 -6287.965} C_VEL
LIN {X 0,Y 495.838,Z 217.719,A -85,B 0,C 180,E1 -6291.03,E2 -6291.03} C_VEL
LIN {X 0,Y 495.879,Z 217.716,A -85,B 0,C 180,E1 -6293.49,E2 -6293.49} C_VEL
LIN {X 0,Y 495.81,Z 217.72,A -85,B 0,C 180,E1 -6296.75,E2 -6296.75} C_VEL
LIN {X 0,Y 495.866,Z 217.709,A -85,B 0,C 180,E1 -6298.376,E2 -6298.376} C_VEL
LIN {X 0,Y 495.963,Z 217.702,A -85,B 0,C 180,E1 -6300.812,E2 -6300.812} C_VEL
LIN {X 0,Y 495.988,Z 217.695,A -85,B 0,C 180,E1 -6302.436,E2 -6302.436} C_VEL
LIN {X 0,Y 495.884,Z 217.716,A -85,B 0,C 180,E1 -6305.694,E2 -6305.694} C_VEL
LIN {X 0,Y 495.834,Z 217.716,A -85,B 0,C 180,E1 -6308.97,E2 -6308.97} C_VEL
LIN {X 0,Y 495.83,Z 217.717,A -85,B 0,C 180,E1 -6312.035,E2 -6312.035} C_VEL
LIN {X 0,Y 495.825,Z 217.726,A -85,B 0,C 180,E1 -6315.451,E2 -6315.451} C_VEL
LIN {X 0,Y 495.78,Z 217.724,A -85,B 0,C 180,E1 -6319.029,E2 -6319.029} C_VEL
LIN {X 0,Y 495.742,Z 217.73,A -85,B 0,C 180,E1 -6321.629,E2 -6321.629} C_VEL
LIN {X 0,Y 495.716,Z 217.731,A -85,B 0,C 180,E1 -6324.277,E2 -6324.277} C_VEL
LIN {X 0,Y 495.784,Z 217.723,A -85,B 0,C 180,E1 -6326.976,E2 -6326.976} C_VEL
LIN {X 0,Y 495.767,Z 217.728,A -85,B 0,C 180,E1 -6329.747,E2 -6329.747} C_VEL
LIN {X 0,Y 495.769,Z 217.725,A -85,B 0,C 180,E1 -6332.595,E2 -6332.595} C_VEL
LIN {X 0,Y 495.747,Z 217.733,A -85,B 0,C 180,E1 -6335.538,E2 -6335.538} C_VEL
LIN {X 0,Y 495.764,Z 217.727,A -85,B 0,C 180,E1 -6338.768,E2 -6338.768} C_VEL
LIN {X 0,Y 495.752,Z 217.731,A -85,B 0,C 180,E1 -6341.782,E2 -6341.782} C_VEL
LIN {X 0,Y 495.739,Z 217.735,A -85,B 0,C 180,E1 -6345.141,E2 -6345.141} C_VEL
LIN {X 0,Y 495.753,Z 217.73,A -85,B 0,C 180,E1 -6348.218,E2 -6348.218} C_VEL
LIN {X 0,Y 495.75,Z 217.738,A -85,B 0,C 180,E1 -6351.408,E2 -6351.408} C_VEL
LIN {X 0,Y 495.748,Z 217.731,A -85,B 0,C 180,E1 -6354.462,E2 -6354.462} C_VEL
LIN {X 0,Y 495.769,Z 217.733,A -85,B 0,C 180,E1 -6357.406,E2 -6357.406} C_VEL
LIN {X 0,Y 495.766,Z 217.725,A -85,B 0,C 180,E1 -6360.254,E2 -6360.254} C_VEL
LIN {X 0,Y 495.74,Z 217.728,A -85,B 0,C 180,E1 -6360.729,E2 -6360.729} C_VEL
LIN {X 0,Y 495.03,Z 217.864,A -85,B 0,C 180,E1 -6361.198,E2 -6361.198} C_VEL
LIN {X 0,Y 489.405,Z 218.597,A -85,B 0,C 180,E1 -6362.644,E2 -6362.644} C_VEL
LIN {X 0,Y 488.924,Z 219.358,A -85,B 0,C 180,E1 -6363.002,E2 -6363.002} C_VEL
LIN {X 0,Y 488.954,Z 219.641,A -85,B 0,C 180,E1 -6363.068,E2 -6363.068} C_VEL
LIN {X 0,Y 489.767,Z 225.571,A -85,B 0,C 180,E1 -6364.273,E2 -6364.273} C_VEL
LIN {X 0,Y 489.403,Z 240.69,A -85,B 0,C 180,E1 -6367.187,E2 -6367.187} C_VEL
LIN {X 0,Y 489.362,Z 243.67,A -85,B 0,C 180,E1 -6367.756,E2 -6367.756} C_VEL
LIN {X 0,Y 491.914,Z 257.623,A -85,B 0,C 180,E1 -6368.06,E2 -6368.06} C_VEL
LIN {X 0,Y 491.175,Z 351.028,A -85,B 0,C 180,E1 -6369.451,E2 -6369.451} C_VEL
LIN {X 0,Y 490.956,Z 364.451,A -85,B 0,C 180,E1 -6369.824,E2 -6369.824} C_VEL
LIN {X 0,Y 490.591,Z 376.708,A -85,B 0,C 180,E1 -6370.327,E2 -6370.327} C_VEL
LIN {X 0,Y 490.301,Z 388.208,A -85,B 0,C 180,E1 -6370.967,E2 -6370.967} C_VEL
LIN {X 0,Y 489.904,Z 398.699,A -85,B 0,C 180,E1 -6371.711,E2 -6371.711} C_VEL
LIN {X 0,Y 489.486,Z 409.489,A -85,B 0,C 180,E1 -6372.667,E2 -6372.667} C_VEL
LIN {X 0,Y 489.063,Z 419.17,A -85,B 0,C 180,E1 -6373.727,E2 -6373.727} C_VEL
LIN {X 0,Y 488.742,Z 426.541,A -85,B 0,C 180,E1 -6374.711,E2 -6374.711} C_VEL
LIN {X 0,Y 488.484,Z 433.571,A -85,B 0,C 180,E1 -6375.843,E2 -6375.843} C_VEL
LIN {X 0,Y 488.3,Z 439.92,A -85,B 0,C 180,E1 -6377.109,E2 -6377.109} C_VEL
LIN {X 0,Y 488.123,Z 444.943,A -85,B 0,C 180,E1 -6378.371,E2 -6378.371} C_VEL
LIN {X 0,Y 488.001,Z 448.81,A -85,B 0,C 180,E1 -6379.629,E2 -6379.629} C_VEL
LIN {X 0,Y 487.891,Z 451.629,A -85,B 0,C 180,E1 -6380.883,E2 -6380.883} C_VEL
LIN {X 0,Y 487.9,Z 452.953,A -85,B 0,C 180,E1 -6381.718,E2 -6381.718} C_VEL
LIN {X 0,Y 487.917,Z 453.88,A -85,B 0,C 180,E1 -6382.551,E2 -6382.551} C_VEL
LIN {X 0,Y 487.922,Z 454.468,A -85,B 0,C 180,E1 -6383.657,E2 -6383.657} C_VEL
LIN {X 0,Y 487.894,Z 454.22,A -85,B 0,C 180,E1 -6385.042,E2 -6385.042} C_VEL
LIN {X 0,Y 487.963,Z 452.485,A -85,B 0,C 180,E1 -6386.697,E2 -6386.697} C_VEL
LIN {X 0,Y 487.969,Z 450.978,A -85,B 0,C 180,E1 -6387.524,E2 -6387.524} C_VEL
LIN {X 0,Y 487.975,Z 447.953,A -85,B 0,C 180,E1 -6388.762,E2 -6388.762} C_VEL
LIN {X 0,Y 488.017,Z 443.893,A -85,B 0,C 180,E1 -6390,E2 -6390} C_VEL
LIN {X 0,Y 488.262,Z 438.671,A -85,B 0,C 180,E1 -6391.237,E2 -6391.237} C_VEL
LIN {X 0,Y 488.447,Z 432.144,A -85,B 0,C 180,E1 -6392.474,E2 -6392.474} C_VEL
LIN {X 0,Y 488.783,Z 424.044,A -85,B 0,C 180,E1 -6393.71,E2 -6393.71} C_VEL
LIN {X 0,Y 489.173,Z 415.768,A -85,B 0,C 180,E1 -6394.739,E2 -6394.739} C_VEL
LIN {X 0,Y 489.58,Z 405.6,A -85,B 0,C 180,E1 -6395.767,E2 -6395.767} C_VEL
LIN {X 0,Y 490.02,Z 394.142,A -85,B 0,C 180,E1 -6396.692,E2 -6396.692} C_VEL
LIN {X 0,Y 490.399,Z 382.853,A -85,B 0,C 180,E1 -6397.411,E2 -6397.411} C_VEL
LIN {X 0,Y 490.76,Z 371.216,A -85,B 0,C 180,E1 -6397.974,E2 -6397.974} C_VEL
LIN {X 0,Y 491.063,Z 357.935,A -85,B 0,C 180,E1 -6398.432,E2 -6398.432} C_VEL
LIN {X 0,Y 491.179,Z 344.68,A -85,B 0,C 180,E1 -6398.716,E2 -6398.716} C_VEL
LIN {X 0,Y 491.742,Z 256.494,A -85,B 0,C 180,E1 -6400.005,E2 -6400.005} C_VEL
LIN {X 0,Y 489.344,Z 243.59,A -85,B 0,C 180,E1 -6400.29,E2 -6400.29} C_VEL
LIN {X 0,Y 489.69,Z 228.038,A -85,B 0,C 180,E1 -6403.275,E2 -6403.275} C_VEL
LIN {X 0,Y 489.679,Z 223.698,A -85,B 0,C 180,E1 -6404.122,E2 -6404.122} C_VEL
LIN {X 0,Y 488.811,Z 218.599,A -85,B 0,C 180,E1 -6405.207,E2 -6405.207} C_VEL
LIN {X 0,Y 488.751,Z 218.607,A -85,B 0,C 180,E1 -6408.442,E2 -6408.442} C_VEL
LIN {X 0,Y 488.71,Z 218.608,A -85,B 0,C 180,E1 -6411.071,E2 -6411.071} C_VEL
LIN {X 0,Y 488.687,Z 218.607,A -85,B 0,C 180,E1 -6413.746,E2 -6413.746} C_VEL
LIN {X 0,Y 488.728,Z 218.607,A -85,B 0,C 180,E1 -6416.928,E2 -6416.928} C_VEL
LIN {X 0,Y 488.727,Z 218.605,A -85,B 0,C 180,E1 -6420.219,E2 -6420.219} C_VEL
LIN {X 0,Y 488.737,Z 218.601,A -85,B 0,C 180,E1 -6423.484,E2 -6423.484} C_VEL
LIN {X 0,Y 488.683,Z 218.612,A -85,B 0,C 180,E1 -6426.354,E2 -6426.354} C_VEL
LIN {X 0,Y 488.702,Z 218.607,A -85,B 0,C 180,E1 -6429.254,E2 -6429.254} C_VEL
LIN {X 0,Y 488.709,Z 218.604,A -85,B 0,C 180,E1 -6431.599,E2 -6431.599} C_VEL
LIN {X 0,Y 488.703,Z 218.612,A -85,B 0,C 180,E1 -6434.802,E2 -6434.802} C_VEL
LIN {X 0,Y 488.69,Z 218.607,A -85,B 0,C 180,E1 -6437.474,E2 -6437.474} C_VEL
LIN {X 0,Y 488.702,Z 218.613,A -85,B 0,C 180,E1 -6440.746,E2 -6440.746} C_VEL
LIN {X 0,Y 488.671,Z 218.609,A -85,B 0,C 180,E1 -6443.867,E2 -6443.867} C_VEL
LIN {X 0,Y 488.74,Z 218.606,A -85,B 0,C 180,E1 -6446.877,E2 -6446.877} C_VEL
LIN {X 0,Y 488.725,Z 218.602,A -85,B 0,C 180,E1 -6449.781,E2 -6449.781} C_VEL
LIN {X 0,Y 488.731,Z 218.61,A -85,B 0,C 180,E1 -6452.602,E2 -6452.602} C_VEL
LIN {X 0,Y 488.699,Z 218.606,A -85,B 0,C 180,E1 -6455.351,E2 -6455.351} C_VEL
LIN {X 0,Y 488.699,Z 218.607,A -85,B 0,C 180,E1 -6458.043,E2 -6458.043} C_VEL
LIN {X 0,Y 488.741,Z 218.608,A -85,B 0,C 180,E1 -6460.686,E2 -6460.686} C_VEL
LIN {X 0,Y 488.761,Z 218.6,A -85,B 0,C 180,E1 -6464.145,E2 -6464.145} C_VEL
LIN {X 0,Y 488.74,Z 218.6,A -85,B 0,C 180,E1 -6467.543,E2 -6467.543} C_VEL
LIN {X 0,Y 488.759,Z 218.6,A -85,B 0,C 180,E1 -6470.064,E2 -6470.064} C_VEL
LIN {X 0,Y 488.825,Z 218.596,A -85,B 0,C 180,E1 -6472.764,E2 -6472.764} C_VEL
LIN {X 0,Y 488.807,Z 218.595,A -85,B 0,C 180,E1 -6475.051,E2 -6475.051} C_VEL
LIN {X 0,Y 488.96,Z 218.573,A -85,B 0,C 180,E1 -6477.529,E2 -6477.529} C_VEL
LIN {X 0,Y 488.934,Z 218.582,A -85,B 0,C 180,E1 -6480.824,E2 -6480.824} C_VEL
LIN {X 0,Y 488.956,Z 218.58,A -85,B 0,C 180,E1 -6482.471,E2 -6482.471} C_VEL
LIN {X 0,Y 488.853,Z 218.586,A -85,B 0,C 180,E1 -6485.776,E2 -6485.776} C_VEL
LIN {X 0,Y 488.816,Z 218.595,A -85,B 0,C 180,E1 -6488.266,E2 -6488.266} C_VEL
LIN {X 0,Y 488.806,Z 218.592,A -85,B 0,C 180,E1 -6491.612,E2 -6491.612} C_VEL
LIN {X 0,Y 488.765,Z 218.6,A -85,B 0,C 180,E1 -6495,E2 -6495} C_VEL
LIN {X 0,Y 488.747,Z 218.606,A -85,B 0,C 180,E1 -6498.442,E2 -6498.442} C_VEL
LIN {X 0,Y 488.707,Z 218.607,A -85,B 0,C 180,E1 -6501.071,E2 -6501.071} C_VEL
LIN {X 0,Y 488.684,Z 218.607,A -85,B 0,C 180,E1 -6503.746,E2 -6503.746} C_VEL
LIN {X 0,Y 488.725,Z 218.606,A -85,B 0,C 180,E1 -6506.928,E2 -6506.928} C_VEL
LIN {X 0,Y 488.724,Z 218.606,A -85,B 0,C 180,E1 -6510.219,E2 -6510.219} C_VEL
LIN {X 0,Y 488.729,Z 218.602,A -85,B 0,C 180,E1 -6513.483,E2 -6513.483} C_VEL
LIN {X 0,Y 488.676,Z 218.614,A -85,B 0,C 180,E1 -6516.353,E2 -6516.353} C_VEL
LIN {X 0,Y 488.698,Z 218.606,A -85,B 0,C 180,E1 -6519.255,E2 -6519.255} C_VEL
LIN {X 0,Y 488.698,Z 218.605,A -85,B 0,C 180,E1 -6521.599,E2 -6521.599} C_VEL
LIN {X 0,Y 488.702,Z 218.61,A -85,B 0,C 180,E1 -6524.803,E2 -6524.803} C_VEL
LIN {X 0,Y 488.689,Z 218.607,A -85,B 0,C 180,E1 -6527.474,E2 -6527.474} C_VEL
LIN {X 0,Y 488.701,Z 218.611,A -85,B 0,C 180,E1 -6530.746,E2 -6530.746} C_VEL
LIN {X 0,Y 488.67,Z 218.61,A -85,B 0,C 180,E1 -6533.867,E2 -6533.867} C_VEL
LIN {X 0,Y 488.74,Z 218.604,A -85,B 0,C 180,E1 -6536.877,E2 -6536.877} C_VEL
LIN {X 0,Y 488.724,Z 218.603,A -85,B 0,C 180,E1 -6539.781,E2 -6539.781} C_VEL
LIN {X 0,Y 488.731,Z 218.61,A -85,B 0,C 180,E1 -6542.602,E2 -6542.602} C_VEL
LIN {X 0,Y 488.706,Z 218.701,A -85,B 0,C 180,E1 -6545.099,E2 -6545.099} C_VEL
LIN {X 0,Y 490.523,Z 228.588,A -85,B 0,C 180,E1 -6546.905,E2 -6546.905} C_VEL
LIN {X 0,Y 490.013,Z 244.634,A -85,B 0,C 180,E1 -6549.647,E2 -6549.647} C_VEL
LIN {X 0,Y 489.411,Z 262.519,A -85,B 0,C 180,E1 -6552.664,E2 -6552.664} C_VEL
LIN {X 0,Y 489.226,Z 269.006,A -85,B 0,C 180,E1 -6553.751,E2 -6553.751} C_VEL
LIN {X 0,Y 491.626,Z 284.838,A -85,B 0,C 180,E1 -6554.064,E2 -6554.064} C_VEL
LIN {X 0,Y 491.07,Z 377.633,A -85,B 0,C 180,E1 -6555.443,E2 -6555.443} C_VEL
LIN {X 0,Y 490.754,Z 390.774,A -85,B 0,C 180,E1 -6555.804,E2 -6555.804} C_VEL
LIN {X 0,Y 490.374,Z 403.442,A -85,B 0,C 180,E1 -6556.321,E2 -6556.321} C_VEL
LIN {X 0,Y 490.004,Z 414.701,A -85,B 0,C 180,E1 -6556.945,E2 -6556.945} C_VEL
LIN {X 0,Y 489.636,Z 425.057,A -85,B 0,C 180,E1 -6557.672,E2 -6557.672} C_VEL
LIN {X 0,Y 489.225,Z 435.766,A -85,B 0,C 180,E1 -6558.608,E2 -6558.608} C_VEL
LIN {X 0,Y 488.839,Z 445.409,A -85,B 0,C 180,E1 -6559.647,E2 -6559.647} C_VEL
LIN {X 0,Y 488.537,Z 453.31,A -85,B 0,C 180,E1 -6560.686,E2 -6560.686} C_VEL
LIN {X 0,Y 488.278,Z 461.024,A -85,B 0,C 180,E1 -6561.933,E2 -6561.933} C_VEL
LIN {X 0,Y 488.096,Z 468.131,A -85,B 0,C 180,E1 -6563.385,E2 -6563.385} C_VEL
LIN {X 0,Y 488.017,Z 472.858,A -85,B 0,C 180,E1 -6564.629,E2 -6564.629} C_VEL
LIN {X 0,Y 487.927,Z 476.466,A -85,B 0,C 180,E1 -6565.87,E2 -6565.87} C_VEL
LIN {X 0,Y 487.964,Z 478.33,A -85,B 0,C 180,E1 -6566.697,E2 -6566.697} C_VEL
LIN {X 0,Y 487.891,Z 480.719,A -85,B 0,C 180,E1 -6568.349,E2 -6568.349} C_VEL
LIN {X 0,Y 487.821,Z 481.54,A -85,B 0,C 180,E1 -6570,E2 -6570} C_VEL
LIN {X 0,Y 487.891,Z 480.717,A -85,B 0,C 180,E1 -6571.651,E2 -6571.651} C_VEL
LIN {X 0,Y 487.964,Z 478.326,A -85,B 0,C 180,E1 -6573.303,E2 -6573.303} C_VEL
LIN {X 0,Y 487.919,Z 475.388,A -85,B 0,C 180,E1 -6574.544,E2 -6574.544} C_VEL
LIN {X 0,Y 488.02,Z 471.417,A -85,B 0,C 180,E1 -6575.786,E2 -6575.786} C_VEL
LIN {X 0,Y 488.18,Z 465.312,A -85,B 0,C 180,E1 -6577.237,E2 -6577.237} C_VEL
LIN {X 0,Y 488.36,Z 458.641,A -85,B 0,C 180,E1 -6578.483,E2 -6578.483} C_VEL
LIN {X 0,Y 488.665,Z 450.368,A -85,B 0,C 180,E1 -6579.729,E2 -6579.729} C_VEL
LIN {X 0,Y 488.997,Z 441.9,A -85,B 0,C 180,E1 -6580.768,E2 -6580.768} C_VEL
LIN {X 0,Y 489.491,Z 431.444,A -85,B 0,C 180,E1 -6581.806,E2 -6581.806} C_VEL
LIN {X 0,Y 489.824,Z 419.768,A -85,B 0,C 180,E1 -6582.738,E2 -6582.738} C_VEL
LIN {X 0,Y 490.279,Z 407.889,A -85,B 0,C 180,E1 -6583.47,E2 -6583.47} C_VEL
LIN {X 0,Y 490.685,Z 395.642,A -85,B 0,C 180,E1 -6584.04,E2 -6584.04} C_VEL
LIN {X 0,Y 491.004,Z 383.139,A -85,B 0,C 180,E1 -6584.453,E2 -6584.453} C_VEL
LIN {X 0,Y 491.204,Z 370.422,A -85,B 0,C 180,E1 -6584.712,E2 -6584.712} C_VEL
LIN {X 0,Y 491.7,Z 284.551,A -85,B 0,C 180,E1 -6585.976,E2 -6585.976} C_VEL
LIN {X 0,Y 489.264,Z 268.868,A -85,B 0,C 180,E1 -6586.309,E2 -6586.309} C_VEL
LIN {X 0,Y 489.873,Z 250.14,A -85,B 0,C 180,E1 -6589.485,E2 -6589.485} C_VEL
LIN {X 0,Y 490.395,Z 234.956,A -85,B 0,C 180,E1 -6592.098,E2 -6592.098} C_VEL
LIN {X 0,Y 490.636,Z 229.011,A -85,B 0,C 180,E1 -6593.131,E2 -6593.131} C_VEL
LIN {X 0,Y 488.697,Z 218.614,A -85,B 0,C 180,E1 -6595.102,E2 -6595.102} C_VEL
LIN {X 0,Y 488.709,Z 218.614,A -85,B 0,C 180,E1 -6597.399,E2 -6597.399} C_VEL
LIN {X 0,Y 488.71,Z 218.607,A -85,B 0,C 180,E1 -6600.362,E2 -6600.362} C_VEL
LIN {X 0,Y 488.736,Z 218.608,A -85,B 0,C 180,E1 -6603.484,E2 -6603.484} C_VEL
LIN {X 0,Y 488.674,Z 218.61,A -85,B 0,C 180,E1 -6606.353,E2 -6606.353} C_VEL
LIN {X 0,Y 488.702,Z 218.612,A -85,B 0,C 180,E1 -6609.254,E2 -6609.254} C_VEL
LIN {X 0,Y 488.689,Z 218.608,A -85,B 0,C 180,E1 -6612.526,E2 -6612.526} C_VEL
LIN {X 0,Y 488.702,Z 218.611,A -85,B 0,C 180,E1 -6615.197,E2 -6615.197} C_VEL
LIN {X 0,Y 488.695,Z 218.607,A -85,B 0,C 180,E1 -6618.583,E2 -6618.583} C_VEL
LIN {X 0,Y 488.701,Z 218.608,A -85,B 0,C 180,E1 -6620.948,E2 -6620.948} C_VEL
LIN {X 0,Y 488.67,Z 218.613,A -85,B 0,C 180,E1 -6623.867,E2 -6623.867} C_VEL
LIN {X 0,Y 488.736,Z 218.6,A -85,B 0,C 180,E1 -6626.877,E2 -6626.877} C_VEL
LIN {X 0,Y 488.725,Z 218.603,A -85,B 0,C 180,E1 -6629.781,E2 -6629.781} C_VEL
LIN {X 0,Y 488.726,Z 218.606,A -85,B 0,C 180,E1 -6633.072,E2 -6633.072} C_VEL
LIN {X 0,Y 488.711,Z 218.608,A -85,B 0,C 180,E1 -6635.352,E2 -6635.352} C_VEL
LIN {X 0,Y 488.699,Z 218.605,A -85,B 0,C 180,E1 -6638.043,E2 -6638.043} C_VEL
LIN {X 0,Y 488.743,Z 218.601,A -85,B 0,C 180,E1 -6640.687,E2 -6640.687} C_VEL
LIN {X 0,Y 488.762,Z 218.598,A -85,B 0,C 180,E1 -6644.145,E2 -6644.145} C_VEL
LIN {X 0,Y 488.733,Z 218.602,A -85,B 0,C 180,E1 -6646.698,E2 -6646.698} C_VEL
LIN {X 0,Y 488.736,Z 218.604,A -85,B 0,C 180,E1 -6649.226,E2 -6649.226} C_VEL
LIN {X 0,Y 488.864,Z 218.583,A -85,B 0,C 180,E1 -6652.566,E2 -6652.566} C_VEL
LIN {X 0,Y 488.81,Z 218.594,A -85,B 0,C 180,E1 -6655.051,E2 -6655.051} C_VEL
LIN {X 0,Y 488.953,Z 218.577,A -85,B 0,C 180,E1 -6657.529,E2 -6657.529} C_VEL
LIN {X 0,Y 488.915,Z 218.58,A -85,B 0,C 180,E1 -6660.824,E2 -6660.824} C_VEL
LIN {X 0,Y 488.955,Z 218.571,A -85,B 0,C 180,E1 -6662.471,E2 -6662.471} C_VEL
LIN {X 0,Y 488.841,Z 218.592,A -85,B 0,C 180,E1 -6665.776,E2 -6665.776} C_VEL
LIN {X 0,Y 488.786,Z 218.591,A -85,B 0,C 180,E1 -6668.267,E2 -6668.267} C_VEL
LIN {X 0,Y 488.807,Z 218.597,A -85,B 0,C 180,E1 -6671.613,E2 -6671.613} C_VEL
LIN {X 0,Y 488.758,Z 218.6,A -85,B 0,C 180,E1 -6675.001,E2 -6675.001} C_VEL
LIN {X 0,Y 488.747,Z 218.596,A -85,B 0,C 180,E1 -6678.443,E2 -6678.443} C_VEL
LIN {X 0,Y 488.708,Z 218.608,A -85,B 0,C 180,E1 -6681.071,E2 -6681.071} C_VEL
LIN {X 0,Y 488.672,Z 218.613,A -85,B 0,C 180,E1 -6683.747,E2 -6683.747} C_VEL
LIN {X 0,Y 488.748,Z 218.599,A -85,B 0,C 180,E1 -6686.933,E2 -6686.933} C_VEL
LIN {X 0,Y 488.723,Z 218.61,A -85,B 0,C 180,E1 -6689.271,E2 -6689.271} C_VEL
LIN {X 0,Y 488.705,Z 218.606,A -85,B 0,C 180,E1 -6692.147,E2 -6692.147} C_VEL
LIN {X 0,Y 488.717,Z 218.608,A -85,B 0,C 180,E1 -6695.115,E2 -6695.115} C_VEL
LIN {X 0,Y 488.678,Z 218.609,A -85,B 0,C 180,E1 -6698.2,E2 -6698.2} C_VEL
LIN {X 0,Y 488.72,Z 218.604,A -85,B 0,C 180,E1 -6700.345,E2 -6700.345} C_VEL
LIN {X 0,Y 488.68,Z 218.615,A -85,B 0,C 180,E1 -6703.656,E2 -6703.656} C_VEL
LIN {X 0,Y 488.678,Z 218.607,A -85,B 0,C 180,E1 -6706.345,E2 -6706.345} C_VEL
LIN {X 0,Y 488.705,Z 218.61,A -85,B 0,C 180,E1 -6709.674,E2 -6709.674} C_VEL
LIN {X 0,Y 488.68,Z 218.613,A -85,B 0,C 180,E1 -6712.841,E2 -6712.841} C_VEL
LIN {X 0,Y 488.726,Z 218.607,A -85,B 0,C 180,E1 -6715.887,E2 -6715.887} C_VEL
LIN {X 0,Y 488.695,Z 218.609,A -85,B 0,C 180,E1 -6718.82,E2 -6718.82} C_VEL
LIN {X 0,Y 488.716,Z 218.607,A -85,B 0,C 180,E1 -6721.669,E2 -6721.669} C_VEL
LIN {X 0,Y 488.769,Z 218.69,A -85,B 0,C 180,E1 -6722.87,E2 -6722.87} C_VEL
LIN {X 0,Y 488.954,Z 219.641,A -85,B 0,C 180,E1 -6723.068,E2 -6723.068} C_VEL
LIN {X 0,Y 488.715,Z 222.695,A -85,B 0,C 180,E1 -6723.658,E2 -6723.658} C_VEL
LIN {X 0,Y 487.388,Z 225.908,A -85,B 0,C 180,E1 -6724.224,E2 -6724.224} C_VEL
LIN {X 0,Y 483.806,Z 232.455,A -85,B 0,C 180,E1 -6725.339,E2 -6725.339} C_VEL
LIN {X 0,Y 482.713,Z 235.694,A -85,B 0,C 180,E1 -6725.924,E2 -6725.924} C_VEL
LIN {X 0,Y 482.604,Z 236.748,A -85,B 0,C 180,E1 -6726.125,E2 -6726.125} C_VEL
LIN {X 0,Y 482.429,Z 244.09,A -85,B 0,C 180,E1 -6727.502,E2 -6727.502} C_VEL
LIN {X 0,Y 485.143,Z 258.021,A -85,B 0,C 180,E1 -6727.818,E2 -6727.818} C_VEL
LIN {X 0,Y 484.336,Z 351.453,A -85,B 0,C 180,E1 -6729.231,E2 -6729.231} C_VEL
LIN {X 0,Y 484.105,Z 364.793,A -85,B 0,C 180,E1 -6729.609,E2 -6729.609} C_VEL
LIN {X 0,Y 483.712,Z 377.575,A -85,B 0,C 180,E1 -6730.146,E2 -6730.146} C_VEL
LIN {X 0,Y 483.363,Z 389.86,A -85,B 0,C 180,E1 -6730.861,E2 -6730.861} C_VEL
LIN {X 0,Y 482.83,Z 401.893,A -85,B 0,C 180,E1 -6731.763,E2 -6731.763} C_VEL
LIN {X 0,Y 482.448,Z 412.092,A -85,B 0,C 180,E1 -6732.734,E2 -6732.734} C_VEL
LIN {X 0,Y 482.052,Z 420.438,A -85,B 0,C 180,E1 -6733.701,E2 -6733.701} C_VEL
LIN {X 0,Y 481.645,Z 429.489,A -85,B 0,C 180,E1 -6734.989,E2 -6734.989} C_VEL
LIN {X 0,Y 481.339,Z 436.738,A -85,B 0,C 180,E1 -6736.275,E2 -6736.275} C_VEL
LIN {X 0,Y 481.206,Z 441.603,A -85,B 0,C 180,E1 -6737.345,E2 -6737.345} C_VEL
LIN {X 0,Y 481.036,Z 446.306,A -85,B 0,C 180,E1 -6738.625,E2 -6738.625} C_VEL
LIN {X 0,Y 480.913,Z 449.875,A -85,B 0,C 180,E1 -6739.9,E2 -6739.9} C_VEL
LIN {X 0,Y 480.805,Z 451.688,A -85,B 0,C 180,E1 -6740.747,E2 -6740.747} C_VEL
LIN {X 0,Y 480.83,Z 454,A -85,B 0,C 180,E1 -6742.441,E2 -6742.441} C_VEL
LIN {X 0,Y 480.848,Z 454.667,A -85,B 0,C 180,E1 -6743.659,E2 -6743.659} C_VEL
LIN {X 0,Y 480.819,Z 454.461,A -85,B 0,C 180,E1 -6744.969,E2 -6744.969} C_VEL
LIN {X 0,Y 480.885,Z 452.794,A -85,B 0,C 180,E1 -6746.649,E2 -6746.649} C_VEL
LIN {X 0,Y 480.878,Z 451.343,A -85,B 0,C 180,E1 -6747.487,E2 -6747.487} C_VEL
LIN {X 0,Y 480.887,Z 448.382,A -85,B 0,C 180,E1 -6748.744,E2 -6748.744} C_VEL
LIN {X 0,Y 480.934,Z 444.388,A -85,B 0,C 180,E1 -6750,E2 -6750} C_VEL
LIN {X 0,Y 481.194,Z 439.238,A -85,B 0,C 180,E1 -6751.255,E2 -6751.255} C_VEL
LIN {X 0,Y 481.384,Z 432.79,A -85,B 0,C 180,E1 -6752.51,E2 -6752.51} C_VEL
LIN {X 0,Y 481.751,Z 424.777,A -85,B 0,C 180,E1 -6753.764,E2 -6753.764} C_VEL
LIN {X 0,Y 482.155,Z 416.605,A -85,B 0,C 180,E1 -6754.808,E2 -6754.808} C_VEL
LIN {X 0,Y 482.579,Z 406.634,A -85,B 0,C 180,E1 -6755.851,E2 -6755.851} C_VEL
LIN {X 0,Y 483.041,Z 395.345,A -85,B 0,C 180,E1 -6756.789,E2 -6756.789} C_VEL
LIN {X 0,Y 483.451,Z 384.29,A -85,B 0,C 180,E1 -6757.518,E2 -6757.518} C_VEL
LIN {X 0,Y 483.855,Z 371.943,A -85,B 0,C 180,E1 -6758.141,E2 -6758.141} C_VEL
LIN {X 0,Y 484.145,Z 359.216,A -85,B 0,C 180,E1 -6758.596,E2 -6758.596} C_VEL
LIN {X 0,Y 484.286,Z 346.373,A -85,B 0,C 180,E1 -6758.889,E2 -6758.889} C_VEL
LIN {X 0,Y 484.856,Z 257.108,A -85,B 0,C 180,E1 -6760.216,E2 -6760.216} C_VEL
LIN {X 0,Y 482.362,Z 243.731,A -85,B 0,C 180,E1 -6760.52,E2 -6760.52} C_VEL
LIN {X 0,Y 482.727,Z 228.517,A -85,B 0,C 180,E1 -6763.47,E2 -6763.47} C_VEL
LIN {X 0,Y 482.596,Z 224.167,A -85,B 0,C 180,E1 -6764.334,E2 -6764.334} C_VEL
LIN {X 0,Y 481.778,Z 219.475,A -85,B 0,C 180,E1 -6765.3,E2 -6765.3} C_VEL
LIN {X 0,Y 481.712,Z 219.485,A -85,B 0,C 180,E1 -6768.722,E2 -6768.722} C_VEL
LIN {X 0,Y 481.649,Z 219.484,A -85,B 0,C 180,E1 -6771.395,E2 -6771.395} C_VEL
LIN {X 0,Y 481.666,Z 219.483,A -85,B 0,C 180,E1 -6774.114,E2 -6774.114} C_VEL
LIN {X 0,Y 481.697,Z 219.48,A -85,B 0,C 180,E1 -6777.127,E2 -6777.127} C_VEL
LIN {X 0,Y 481.676,Z 219.48,A -85,B 0,C 180,E1 -6779.741,E2 -6779.741} C_VEL
LIN {X 0,Y 481.674,Z 219.489,A -85,B 0,C 180,E1 -6782.674,E2 -6782.674} C_VEL
LIN {X 0,Y 481.638,Z 219.485,A -85,B 0,C 180,E1 -6785.709,E2 -6785.709} C_VEL
LIN {X 0,Y 481.672,Z 219.487,A -85,B 0,C 180,E1 -6788.859,E2 -6788.859} C_VEL
LIN {X 0,Y 481.654,Z 219.483,A -85,B 0,C 180,E1 -6791.913,E2 -6791.913} C_VEL
LIN {X 0,Y 481.656,Z 219.488,A -85,B 0,C 180,E1 -6794.458,E2 -6794.458} C_VEL
LIN {X 0,Y 481.645,Z 219.484,A -85,B 0,C 180,E1 -6797.839,E2 -6797.839} C_VEL
LIN {X 0,Y 481.662,Z 219.491,A -85,B 0,C 180,E1 -6800.654,E2 -6800.654} C_VEL
LIN {X 0,Y 481.623,Z 219.488,A -85,B 0,C 180,E1 -6803.377,E2 -6803.377} C_VEL
LIN {X 0,Y 481.711,Z 219.48,A -85,B 0,C 180,E1 -6806.33,E2 -6806.33} C_VEL
LIN {X 0,Y 481.652,Z 219.484,A -85,B 0,C 180,E1 -6809.417,E2 -6809.417} C_VEL
LIN {X 0,Y 481.692,Z 219.481,A -85,B 0,C 180,E1 -6812.167,E2 -6812.167} C_VEL
LIN {X 0,Y 481.677,Z 219.484,A -85,B 0,C 180,E1 -6814.967,E2 -6814.967} C_VEL
LIN {X 0,Y 481.649,Z 219.484,A -85,B 0,C 180,E1 -6817.705,E2 -6817.705} C_VEL
LIN {X 0,Y 481.704,Z 219.482,A -85,B 0,C 180,E1 -6820.393,E2 -6820.393} C_VEL
LIN {X 0,Y 481.676,Z 219.483,A -85,B 0,C 180,E1 -6823.033,E2 -6823.033} C_VEL
LIN {X 0,Y 481.683,Z 219.479,A -85,B 0,C 180,E1 -6825.638,E2 -6825.638} C_VEL
LIN {X 0,Y 481.752,Z 219.474,A -85,B 0,C 180,E1 -6828.215,E2 -6828.215} C_VEL
LIN {X 0,Y 481.74,Z 219.472,A -85,B 0,C 180,E1 -6831.611,E2 -6831.611} C_VEL
LIN {X 0,Y 481.8,Z 219.467,A -85,B 0,C 180,E1 -6834.139,E2 -6834.139} C_VEL
LIN {X 0,Y 481.927,Z 219.449,A -85,B 0,C 180,E1 -6837.492,E2 -6837.492} C_VEL
LIN {X 0,Y 481.886,Z 219.46,A -85,B 0,C 180,E1 -6840.836,E2 -6840.836} C_VEL
LIN {X 0,Y 481.922,Z 219.457,A -85,B 0,C 180,E1 -6842.507,E2 -6842.507} C_VEL
LIN {X 0,Y 481.815,Z 219.464,A -85,B 0,C 180,E1 -6845.86,E2 -6845.86} C_VEL
LIN {X 0,Y 481.762,Z 219.475,A -85,B 0,C 180,E1 -6848.388,E2 -6848.388} C_VEL
LIN {X 0,Y 481.751,Z 219.471,A -85,B 0,C 180,E1 -6851.785,E2 -6851.785} C_VEL
LIN {X 0,Y 481.745,Z 219.473,A -85,B 0,C 180,E1 -6855.224,E2 -6855.224} C_VEL
LIN {X 0,Y 481.709,Z 219.483,A -85,B 0,C 180,E1 -6858.722,E2 -6858.722} C_VEL
LIN {X 0,Y 481.646,Z 219.484,A -85,B 0,C 180,E1 -6861.395,E2 -6861.395} C_VEL
LIN {X 0,Y 481.664,Z 219.484,A -85,B 0,C 180,E1 -6864.114,E2 -6864.114} C_VEL
LIN {X 0,Y 481.695,Z 219.48,A -85,B 0,C 180,E1 -6867.127,E2 -6867.127} C_VEL
LIN {X 0,Y 481.674,Z 219.481,A -85,B 0,C 180,E1 -6869.742,E2 -6869.742} C_VEL
LIN {X 0,Y 481.671,Z 219.488,A -85,B 0,C 180,E1 -6872.674,E2 -6872.674} C_VEL
LIN {X 0,Y 481.633,Z 219.486,A -85,B 0,C 180,E1 -6875.71,E2 -6875.71} C_VEL
LIN {X 0,Y 481.668,Z 219.486,A -85,B 0,C 180,E1 -6878.859,E2 -6878.859} C_VEL
LIN {X 0,Y 481.647,Z 219.485,A -85,B 0,C 180,E1 -6881.912,E2 -6881.912} C_VEL
LIN {X 0,Y 481.654,Z 219.49,A -85,B 0,C 180,E1 -6884.458,E2 -6884.458} C_VEL
LIN {X 0,Y 481.644,Z 219.485,A -85,B 0,C 180,E1 -6887.839,E2 -6887.839} C_VEL
LIN {X 0,Y 481.661,Z 219.489,A -85,B 0,C 180,E1 -6890.654,E2 -6890.654} C_VEL
LIN {X 0,Y 481.623,Z 219.487,A -85,B 0,C 180,E1 -6893.377,E2 -6893.377} C_VEL
LIN {X 0,Y 481.711,Z 219.482,A -85,B 0,C 180,E1 -6896.33,E2 -6896.33} C_VEL
LIN {X 0,Y 481.651,Z 219.484,A -85,B 0,C 180,E1 -6899.418,E2 -6899.418} C_VEL
LIN {X 0,Y 481.693,Z 219.484,A -85,B 0,C 180,E1 -6902.168,E2 -6902.168} C_VEL
LIN {X 0,Y 481.688,Z 219.517,A -85,B 0,C 180,E1 -6904.918,E2 -6904.918} C_VEL
LIN {X 0,Y 483.558,Z 230.207,A -85,B 0,C 180,E1 -6906.895,E2 -6906.895} C_VEL
LIN {X 0,Y 482.952,Z 246.885,A -85,B 0,C 180,E1 -6909.781,E2 -6909.781} C_VEL
LIN {X 0,Y 482.389,Z 263.499,A -85,B 0,C 180,E1 -6912.622,E2 -6912.622} C_VEL
LIN {X 0,Y 482.233,Z 268.783,A -85,B 0,C 180,E1 -6913.521,E2 -6913.521} C_VEL
LIN {X 0,Y 484.762,Z 286.131,A -85,B 0,C 180,E1 -6913.869,E2 -6913.869} C_VEL
LIN {X 0,Y 484.195,Z 376.871,A -85,B 0,C 180,E1 -6915.231,E2 -6915.231} C_VEL
LIN {X 0,Y 483.863,Z 390.211,A -85,B 0,C 180,E1 -6915.597,E2 -6915.597} C_VEL
LIN {X 0,Y 483.467,Z 402.986,A -85,B 0,C 180,E1 -6916.122,E2 -6916.122} C_VEL
LIN {X 0,Y 483.071,Z 414.327,A -85,B 0,C 180,E1 -6916.754,E2 -6916.754} C_VEL
LIN {X 0,Y 482.632,Z 424.644,A -85,B 0,C 180,E1 -6917.484,E2 -6917.484} C_VEL
LIN {X 0,Y 482.249,Z 435.461,A -85,B 0,C 180,E1 -6918.441,E2 -6918.441} C_VEL
LIN {X 0,Y 481.82,Z 445.127,A -85,B 0,C 180,E1 -6919.495,E2 -6919.495} C_VEL
LIN {X 0,Y 481.484,Z 453.05,A -85,B 0,C 180,E1 -6920.549,E2 -6920.549} C_VEL
LIN {X 0,Y 481.228,Z 460.784,A -85,B 0,C 180,E1 -6921.814,E2 -6921.814} C_VEL
LIN {X 0,Y 481.012,Z 467.901,A -85,B 0,C 180,E1 -6923.288,E2 -6923.288} C_VEL
LIN {X 0,Y 480.93,Z 472.638,A -85,B 0,C 180,E1 -6924.549,E2 -6924.549} C_VEL
LIN {X 0,Y 480.827,Z 476.254,A -85,B 0,C 180,E1 -6925.809,E2 -6925.809} C_VEL
LIN {X 0,Y 480.888,Z 478.123,A -85,B 0,C 180,E1 -6926.649,E2 -6926.649} C_VEL
LIN {X 0,Y 480.823,Z 479.521,A -85,B 0,C 180,E1 -6927.487,E2 -6927.487} C_VEL
LIN {X 0,Y 480.76,Z 481.126,A -85,B 0,C 180,E1 -6929.162,E2 -6929.162} C_VEL
LIN {X 0,Y 480.745,Z 481.344,A -85,B 0,C 180,E1 -6930,E2 -6930} C_VEL
LIN {X 0,Y 480.76,Z 481.131,A -85,B 0,C 180,E1 -6930.838,E2 -6930.838} C_VEL
LIN {X 0,Y 480.823,Z 479.532,A -85,B 0,C 180,E1 -6932.513,E2 -6932.513} C_VEL
LIN {X 0,Y 480.888,Z 478.141,A -85,B 0,C 180,E1 -6933.351,E2 -6933.351} C_VEL
LIN {X 0,Y 480.838,Z 475.208,A -85,B 0,C 180,E1 -6934.611,E2 -6934.611} C_VEL
LIN {X 0,Y 480.925,Z 471.243,A -85,B 0,C 180,E1 -6935.871,E2 -6935.871} C_VEL
LIN {X 0,Y 481.105,Z 465.152,A -85,B 0,C 180,E1 -6937.344,E2 -6937.344} C_VEL
LIN {X 0,Y 481.318,Z 458.495,A -85,B 0,C 180,E1 -6938.608,E2 -6938.608} C_VEL
LIN {X 0,Y 481.641,Z 450.242,A -85,B 0,C 180,E1 -6939.872,E2 -6939.872} C_VEL
LIN {X 0,Y 482.017,Z 441.797,A -85,B 0,C 180,E1 -6940.926,E2 -6940.926} C_VEL
LIN {X 0,Y 482.534,Z 431.393,A -85,B 0,C 180,E1 -6941.977,E2 -6941.977} C_VEL
LIN {X 0,Y 482.869,Z 420.145,A -85,B 0,C 180,E1 -6942.894,E2 -6942.894} C_VEL
LIN {X 0,Y 483.364,Z 407.936,A -85,B 0,C 180,E1 -6943.667,E2 -6943.667} C_VEL
LIN {X 0,Y 483.806,Z 395.773,A -85,B 0,C 180,E1 -6944.243,E2 -6944.243} C_VEL
LIN {X 0,Y 484.178,Z 382.498,A -85,B 0,C 180,E1 -6944.689,E2 -6944.689} C_VEL
LIN {X 0,Y 484.399,Z 369.37,A -85,B 0,C 180,E1 -6944.95,E2 -6944.95} C_VEL
LIN {X 0,Y 484.926,Z 285.382,A -85,B 0,C 180,E1 -6946.205,E2 -6946.205} C_VEL
LIN {X 0,Y 482.282,Z 268.698,A -85,B 0,C 180,E1 -6946.564,E2 -6946.564} C_VEL
LIN {X 0,Y 482.973,Z 250.053,A -85,B 0,C 180,E1 -6949.775,E2 -6949.775} C_VEL
LIN {X 0,Y 483.648,Z 233.619,A -85,B 0,C 180,E1 -6952.649,E2 -6952.649} C_VEL
LIN {X 0,Y 483.537,Z 228.841,A -85,B 0,C 180,E1 -6953.509,E2 -6953.509} C_VEL
LIN {X 0,Y 481.658,Z 219.492,A -85,B 0,C 180,E1 -6955.338,E2 -6955.338} C_VEL
LIN {X 0,Y 481.67,Z 219.489,A -85,B 0,C 180,E1 -6957.834,E2 -6957.834} C_VEL
LIN {X 0,Y 481.646,Z 219.487,A -85,B 0,C 180,E1 -6960.711,E2 -6960.711} C_VEL
LIN {X 0,Y 481.699,Z 219.484,A -85,B 0,C 180,E1 -6963.733,E2 -6963.733} C_VEL
LIN {X 0,Y 481.621,Z 219.489,A -85,B 0,C 180,E1 -6966.747,E2 -6966.747} C_VEL
LIN {X 0,Y 481.669,Z 219.485,A -85,B 0,C 180,E1 -6969.941,E2 -6969.941} C_VEL
LIN {X 0,Y 481.629,Z 219.492,A -85,B 0,C 180,E1 -6973.146,E2 -6973.146} C_VEL
LIN {X 0,Y 481.653,Z 219.49,A -85,B 0,C 180,E1 -6975.641,E2 -6975.641} C_VEL
LIN {X 0,Y 481.65,Z 219.487,A -85,B 0,C 180,E1 -6978.957,E2 -6978.957} C_VEL
LIN {X 0,Y 481.65,Z 219.485,A -85,B 0,C 180,E1 -6981.994,E2 -6981.994} C_VEL
LIN {X 0,Y 481.684,Z 219.486,A -85,B 0,C 180,E1 -6985.317,E2 -6985.317} C_VEL
LIN {X 0,Y 481.645,Z 219.485,A -85,B 0,C 180,E1 -6988.312,E2 -6988.312} C_VEL
LIN {X 0,Y 481.675,Z 219.483,A -85,B 0,C 180,E1 -6991.217,E2 -6991.217} C_VEL
LIN {X 0,Y 481.669,Z 219.48,A -85,B 0,C 180,E1 -6994.041,E2 -6994.041} C_VEL
LIN {X 0,Y 481.675,Z 219.482,A -85,B 0,C 180,E1 -6996.812,E2 -6996.812} C_VEL
LIN {X 0,Y 481.696,Z 219.484,A -85,B 0,C 180,E1 -6999.503,E2 -6999.503} C_VEL
LIN {X 0,Y 481.692,Z 219.478,A -85,B 0,C 180,E1 -7002.158,E2 -7002.158} C_VEL
LIN {X 0,Y 481.745,Z 219.472,A -85,B 0,C 180,E1 -7004.776,E2 -7004.776} C_VEL
LIN {X 0,Y 481.752,Z 219.468,A -85,B 0,C 180,E1 -7008.215,E2 -7008.215} C_VEL
LIN {X 0,Y 481.762,Z 219.473,A -85,B 0,C 180,E1 -7011.612,E2 -7011.612} C_VEL
LIN {X 0,Y 481.815,Z 219.463,A -85,B 0,C 180,E1 -7014.14,E2 -7014.14} C_VEL
LIN {X 0,Y 481.919,Z 219.453,A -85,B 0,C 180,E1 -7017.493,E2 -7017.493} C_VEL
LIN {X 0,Y 481.941,Z 219.449,A -85,B 0,C 180,E1 -7020,E2 -7020} C_VEL
LIN {X 0,Y 481.921,Z 219.448,A -85,B 0,C 180,E1 -7022.508,E2 -7022.508} C_VEL
LIN {X 0,Y 481.8,Z 219.468,A -85,B 0,C 180,E1 -7025.861,E2 -7025.861} C_VEL
LIN {X 0,Y 481.74,Z 219.468,A -85,B 0,C 180,E1 -7028.389,E2 -7028.389} C_VEL
LIN {X 0,Y 481.752,Z 219.473,A -85,B 0,C 180,E1 -7031.785,E2 -7031.785} C_VEL
LIN {X 0,Y 481.741,Z 219.477,A -85,B 0,C 180,E1 -7035.224,E2 -7035.224} C_VEL
LIN {X 0,Y 481.708,Z 219.474,A -85,B 0,C 180,E1 -7038.722,E2 -7038.722} C_VEL
LIN {X 0,Y 481.647,Z 219.49,A -85,B 0,C 180,E1 -7041.395,E2 -7041.395} C_VEL
LIN {X 0,Y 481.651,Z 219.484,A -85,B 0,C 180,E1 -7044.115,E2 -7044.115} C_VEL
LIN {X 0,Y 481.716,Z 219.477,A -85,B 0,C 180,E1 -7047.132,E2 -7047.132} C_VEL
LIN {X 0,Y 481.679,Z 219.483,A -85,B 0,C 180,E1 -7049.741,E2 -7049.741} C_VEL
LIN {X 0,Y 481.674,Z 219.482,A -85,B 0,C 180,E1 -7052.674,E2 -7052.674} C_VEL
LIN {X 0,Y 481.662,Z 219.488,A -85,B 0,C 180,E1 -7055.204,E2 -7055.204} C_VEL
LIN {X 0,Y 481.672,Z 219.483,A -85,B 0,C 180,E1 -7058.859,E2 -7058.859} C_VEL
LIN {X 0,Y 481.649,Z 219.487,A -85,B 0,C 180,E1 -7061.912,E2 -7061.912} C_VEL
LIN {X 0,Y 481.656,Z 219.485,A -85,B 0,C 180,E1 -7064.458,E2 -7064.458} C_VEL
LIN {X 0,Y 481.645,Z 219.491,A -85,B 0,C 180,E1 -7067.839,E2 -7067.839} C_VEL
LIN {X 0,Y 481.659,Z 219.484,A -85,B 0,C 180,E1 -7070.655,E2 -7070.655} C_VEL
LIN {X 0,Y 481.629,Z 219.497,A -85,B 0,C 180,E1 -7073.377,E2 -7073.377} C_VEL
LIN {X 0,Y 481.679,Z 219.482,A -85,B 0,C 180,E1 -7076.328,E2 -7076.328} C_VEL
LIN {X 0,Y 481.654,Z 219.488,A -85,B 0,C 180,E1 -7079.418,E2 -7079.418} C_VEL
LIN {X 0,Y 481.711,Z 219.553,A -85,B 0,C 180,E1 -7082.679,E2 -7082.679} C_VEL
LIN {X 0,Y 482.821,Z 226.44,A -85,B 0,C 180,E1 -7084.108,E2 -7084.108} C_VEL
LIN {X 0,Y 482.604,Z 236.748,A -85,B 0,C 180,E1 -7086.125,E2 -7086.125} C_VEL
LIN {X 0,Y 481.983,Z 239.202,A -85,B 0,C 180,E1 -7086.51,E2 -7086.51} C_VEL
LIN {X 0,Y 480.644,Z 242.101,A -85,B 0,C 180,E1 -7086.828,E2 -7086.828} C_VEL
LIN {X 0,Y 478.649,Z 246.49,A -85,B 0,C 180,E1 -7087.159,E2 -7087.159} C_VEL
LIN {X 0,Y 477.489,Z 250.818,A -85,B 0,C 180,E1 -7087.367,E2 -7087.367} C_VEL
LIN {X 0,Y 477.495,Z 254.111,A -85,B 0,C 180,E1 -7087.465,E2 -7087.465} C_VEL
LIN {X 0,Y 478.391,Z 259.774,A -85,B 0,C 180,E1 -7087.588,E2 -7087.588} C_VEL
LIN {X 0,Y 477.513,Z 352.005,A -85,B 0,C 180,E1 -7089.005,E2 -7089.005} C_VEL
LIN {X 0,Y 477.277,Z 365.223,A -85,B 0,C 180,E1 -7089.389,E2 -7089.389} C_VEL
LIN {X 0,Y 476.89,Z 377.371,A -85,B 0,C 180,E1 -7089.906,E2 -7089.906} C_VEL
LIN {X 0,Y 476.526,Z 388.48,A -85,B 0,C 180,E1 -7090.542,E2 -7090.542} C_VEL
LIN {X 0,Y 476.047,Z 399.882,A -85,B 0,C 180,E1 -7091.382,E2 -7091.382} C_VEL
LIN {X 0,Y 475.568,Z 410.526,A -85,B 0,C 180,E1 -7092.365,E2 -7092.365} C_VEL
LIN {X 0,Y 475.081,Z 420.062,A -85,B 0,C 180,E1 -7093.455,E2 -7093.455} C_VEL
LIN {X 0,Y 474.655,Z 429.205,A -85,B 0,C 180,E1 -7094.763,E2 -7094.763} C_VEL
LIN {X 0,Y 474.313,Z 436.541,A -85,B 0,C 180,E1 -7096.067,E2 -7096.067} C_VEL
LIN {X 0,Y 474.17,Z 441.477,A -85,B 0,C 180,E1 -7097.154,E2 -7097.154} C_VEL
LIN {X 0,Y 473.988,Z 446.409,A -85,B 0,C 180,E1 -7098.502,E2 -7098.502} C_VEL
LIN {X 0,Y 473.829,Z 449.88,A -85,B 0,C 180,E1 -7099.747,E2 -7099.747} C_VEL
LIN {X 0,Y 473.724,Z 451.747,A -85,B 0,C 180,E1 -7100.608,E2 -7100.608} C_VEL
LIN {X 0,Y 473.727,Z 453.138,A -85,B 0,C 180,E1 -7101.468,E2 -7101.468} C_VEL
LIN {X 0,Y 473.757,Z 454.723,A -85,B 0,C 180,E1 -7103.184,E2 -7103.184} C_VEL
LIN {X 0,Y 473.736,Z 454.928,A -85,B 0,C 180,E1 -7104.039,E2 -7104.039} C_VEL
LIN {X 0,Y 473.745,Z 454.701,A -85,B 0,C 180,E1 -7104.893,E2 -7104.893} C_VEL
LIN {X 0,Y 473.789,Z 453.091,A -85,B 0,C 180,E1 -7106.598,E2 -7106.598} C_VEL
LIN {X 0,Y 473.791,Z 451.696,A -85,B 0,C 180,E1 -7107.449,E2 -7107.449} C_VEL
LIN {X 0,Y 473.804,Z 448.785,A -85,B 0,C 180,E1 -7108.725,E2 -7108.725} C_VEL
LIN {X 0,Y 473.85,Z 444.852,A -85,B 0,C 180,E1 -7110,E2 -7110} C_VEL
LIN {X 0,Y 474.127,Z 439.78,A -85,B 0,C 180,E1 -7111.274,E2 -7111.274} C_VEL
LIN {X 0,Y 474.319,Z 433.417,A -85,B 0,C 180,E1 -7112.548,E2 -7112.548} C_VEL
LIN {X 0,Y 474.72,Z 425.489,A -85,B 0,C 180,E1 -7113.82,E2 -7113.82} C_VEL
LIN {X 0,Y 475.136,Z 417.416,A -85,B 0,C 180,E1 -7114.879,E2 -7114.879} C_VEL
LIN {X 0,Y 475.573,Z 407.588,A -85,B 0,C 180,E1 -7115.938,E2 -7115.938} C_VEL
LIN {X 0,Y 476.063,Z 396.51,A -85,B 0,C 180,E1 -7116.889,E2 -7116.889} C_VEL
LIN {X 0,Y 476.478,Z 385.684,A -85,B 0,C 180,E1 -7117.628,E2 -7117.628} C_VEL
LIN {X 0,Y 476.888,Z 373.726,A -85,B 0,C 180,E1 -7118.261,E2 -7118.261} C_VEL
LIN {X 0,Y 477.229,Z 361.155,A -85,B 0,C 180,E1 -7118.743,E2 -7118.743} C_VEL
LIN {X 0,Y 477.42,Z 348.008,A -85,B 0,C 180,E1 -7119.065,E2 -7119.065} C_VEL
LIN {X 0,Y 477.961,Z 257.788,A -85,B 0,C 180,E1 -7120.431,E2 -7120.431} C_VEL
LIN {X 0,Y 475.389,Z 244,A -85,B 0,C 180,E1 -7120.73,E2 -7120.73} C_VEL
LIN {X 0,Y 475.77,Z 228.992,A -85,B 0,C 180,E1 -7123.671,E2 -7123.671} C_VEL
LIN {X 0,Y 475.463,Z 224.636,A -85,B 0,C 180,E1 -7124.553,E2 -7124.553} C_VEL
LIN {X 0,Y 474.729,Z 220.352,A -85,B 0,C 180,E1 -7125.455,E2 -7125.455} C_VEL
LIN {X 0,Y 474.666,Z 220.36,A -85,B 0,C 180,E1 -7129.01,E2 -7129.01} C_VEL
LIN {X 0,Y 474.592,Z 220.363,A -85,B 0,C 180,E1 -7131.729,E2 -7131.729} C_VEL
LIN {X 0,Y 474.644,Z 220.362,A -85,B 0,C 180,E1 -7134.494,E2 -7134.494} C_VEL
LIN {X 0,Y 474.639,Z 220.358,A -85,B 0,C 180,E1 -7137.324,E2 -7137.324} C_VEL
LIN {X 0,Y 474.606,Z 220.364,A -85,B 0,C 180,E1 -7140.23,E2 -7140.23} C_VEL
LIN {X 0,Y 474.645,Z 220.358,A -85,B 0,C 180,E1 -7143.22,E2 -7143.22} C_VEL
LIN {X 0,Y 474.59,Z 220.367,A -85,B 0,C 180,E1 -7146.323,E2 -7146.323} C_VEL
LIN {X 0,Y 474.62,Z 220.359,A -85,B 0,C 180,E1 -7149.646,E2 -7149.646} C_VEL
LIN {X 0,Y 474.616,Z 220.365,A -85,B 0,C 180,E1 -7152.934,E2 -7152.934} C_VEL
LIN {X 0,Y 474.605,Z 220.362,A -85,B 0,C 180,E1 -7155.894,E2 -7155.894} C_VEL
LIN {X 0,Y 474.624,Z 220.362,A -85,B 0,C 180,E1 -7159.041,E2 -7159.041} C_VEL
LIN {X 0,Y 474.609,Z 220.361,A -85,B 0,C 180,E1 -7161.704,E2 -7161.704} C_VEL
LIN {X 0,Y 474.623,Z 220.367,A -85,B 0,C 180,E1 -7164.725,E2 -7164.725} C_VEL
LIN {X 0,Y 474.637,Z 220.357,A -85,B 0,C 180,E1 -7167.788,E2 -7167.788} C_VEL
LIN {X 0,Y 474.623,Z 220.364,A -85,B 0,C 180,E1 -7170.885,E2 -7170.885} C_VEL
LIN {X 0,Y 474.627,Z 220.358,A -85,B 0,C 180,E1 -7173.626,E2 -7173.626} C_VEL
LIN {X 0,Y 474.635,Z 220.366,A -85,B 0,C 180,E1 -7176.642,E2 -7176.642} C_VEL
LIN {X 0,Y 474.654,Z 220.357,A -85,B 0,C 180,E1 -7180.089,E2 -7180.089} C_VEL
LIN {X 0,Y 474.636,Z 220.364,A -85,B 0,C 180,E1 -7182.774,E2 -7182.774} C_VEL
LIN {X 0,Y 474.643,Z 220.357,A -85,B 0,C 180,E1 -7185.421,E2 -7185.421} C_VEL
LIN {X 0,Y 474.705,Z 220.35,A -85,B 0,C 180,E1 -7188.037,E2 -7188.037} C_VEL
LIN {X 0,Y 474.712,Z 220.348,A -85,B 0,C 180,E1 -7191.486,E2 -7191.486} C_VEL
LIN {X 0,Y 474.747,Z 220.348,A -85,B 0,C 180,E1 -7194.904,E2 -7194.904} C_VEL
LIN {X 0,Y 474.893,Z 220.325,A -85,B 0,C 180,E1 -7197.455,E2 -7197.455} C_VEL
LIN {X 0,Y 474.911,Z 220.324,A -85,B 0,C 180,E1 -7200,E2 -7200} C_VEL
LIN {X 0,Y 474.887,Z 220.334,A -85,B 0,C 180,E1 -7202.545,E2 -7202.545} C_VEL
LIN {X 0,Y 474.778,Z 220.341,A -85,B 0,C 180,E1 -7205.948,E2 -7205.948} C_VEL
LIN {X 0,Y 474.727,Z 220.353,A -85,B 0,C 180,E1 -7208.513,E2 -7208.513} C_VEL
LIN {X 0,Y 474.705,Z 220.35,A -85,B 0,C 180,E1 -7211.962,E2 -7211.962} C_VEL
LIN {X 0,Y 474.701,Z 220.349,A -85,B 0,C 180,E1 -7215.456,E2 -7215.456} C_VEL
LIN {X 0,Y 474.663,Z 220.357,A -85,B 0,C 180,E1 -7219.01,E2 -7219.01} C_VEL
LIN {X 0,Y 474.589,Z 220.363,A -85,B 0,C 180,E1 -7221.729,E2 -7221.729} C_VEL
LIN {X 0,Y 474.641,Z 220.364,A -85,B 0,C 180,E1 -7224.494,E2 -7224.494} C_VEL
LIN {X 0,Y 474.637,Z 220.358,A -85,B 0,C 180,E1 -7227.324,E2 -7227.324} C_VEL
LIN {X 0,Y 474.603,Z 220.365,A -85,B 0,C 180,E1 -7230.23,E2 -7230.23} C_VEL
LIN {X 0,Y 474.625,Z 220.36,A -85,B 0,C 180,E1 -7233.222,E2 -7233.222} C_VEL
LIN {X 0,Y 474.585,Z 220.369,A -85,B 0,C 180,E1 -7236.324,E2 -7236.324} C_VEL
LIN {X 0,Y 474.624,Z 220.359,A -85,B 0,C 180,E1 -7239.548,E2 -7239.548} C_VEL
LIN {X 0,Y 474.6,Z 220.366,A -85,B 0,C 180,E1 -7242.233,E2 -7242.233} C_VEL
LIN {X 0,Y 474.617,Z 220.36,A -85,B 0,C 180,E1 -7245.298,E2 -7245.298} C_VEL
LIN {X 0,Y 474.616,Z 220.364,A -85,B 0,C 180,E1 -7248.214,E2 -7248.214} C_VEL
LIN {X 0,Y 474.611,Z 220.36,A -85,B 0,C 180,E1 -7251.543,E2 -7251.543} C_VEL
LIN {X 0,Y 474.623,Z 220.365,A -85,B 0,C 180,E1 -7254.726,E2 -7254.726} C_VEL
LIN {X 0,Y 474.637,Z 220.358,A -85,B 0,C 180,E1 -7257.788,E2 -7257.788} C_VEL
LIN {X 0,Y 474.623,Z 220.364,A -85,B 0,C 180,E1 -7260.885,E2 -7260.885} C_VEL
LIN {X 0,Y 474.628,Z 220.363,A -85,B 0,C 180,E1 -7263.626,E2 -7263.626} C_VEL
LIN {X 0,Y 474.634,Z 220.41,A -85,B 0,C 180,E1 -7264.746,E2 -7264.746} C_VEL
LIN {X 0,Y 476.585,Z 231.159,A -85,B 0,C 180,E1 -7266.767,E2 -7266.767} C_VEL
LIN {X 0,Y 476.056,Z 246.566,A -85,B 0,C 180,E1 -7269.475,E2 -7269.475} C_VEL
LIN {X 0,Y 475.374,Z 264.468,A -85,B 0,C 180,E1 -7272.58,E2 -7272.58} C_VEL
LIN {X 0,Y 475.27,Z 268.898,A -85,B 0,C 180,E1 -7273.302,E2 -7273.302} C_VEL
LIN {X 0,Y 477.892,Z 286.337,A -85,B 0,C 180,E1 -7273.654,E2 -7273.654} C_VEL
LIN {X 0,Y 477.309,Z 377.135,A -85,B 0,C 180,E1 -7275.041,E2 -7275.041} C_VEL
LIN {X 0,Y 476.947,Z 390.324,A -85,B 0,C 180,E1 -7275.411,E2 -7275.411} C_VEL
LIN {X 0,Y 476.529,Z 402.455,A -85,B 0,C 180,E1 -7275.916,E2 -7275.916} C_VEL
LIN {X 0,Y 476.109,Z 414.221,A -85,B 0,C 180,E1 -7276.578,E2 -7276.578} C_VEL
LIN {X 0,Y 475.616,Z 425.326,A -85,B 0,C 180,E1 -7277.385,E2 -7277.385} C_VEL
LIN {X 0,Y 475.216,Z 436.197,A -85,B 0,C 180,E1 -7278.375,E2 -7278.375} C_VEL
LIN {X 0,Y 474.783,Z 444.814,A -85,B 0,C 180,E1 -7279.337,E2 -7279.337} C_VEL
LIN {X 0,Y 474.457,Z 452.76,A -85,B 0,C 180,E1 -7280.407,E2 -7280.407} C_VEL
LIN {X 0,Y 474.164,Z 460.522,A -85,B 0,C 180,E1 -7281.691,E2 -7281.691} C_VEL
LIN {X 0,Y 473.925,Z 467.655,A -85,B 0,C 180,E1 -7283.187,E2 -7283.187} C_VEL
LIN {X 0,Y 473.844,Z 472.404,A -85,B 0,C 180,E1 -7284.468,E2 -7284.468} C_VEL
LIN {X 0,Y 473.733,Z 476.03,A -85,B 0,C 180,E1 -7285.746,E2 -7285.746} C_VEL
LIN {X 0,Y 473.795,Z 477.906,A -85,B 0,C 180,E1 -7286.598,E2 -7286.598} C_VEL
LIN {X 0,Y 473.741,Z 479.311,A -85,B 0,C 180,E1 -7287.449,E2 -7287.449} C_VEL
LIN {X 0,Y 473.688,Z 480.925,A -85,B 0,C 180,E1 -7289.15,E2 -7289.15} C_VEL
LIN {X 0,Y 473.671,Z 481.148,A -85,B 0,C 180,E1 -7290,E2 -7290} C_VEL
LIN {X 0,Y 473.688,Z 480.941,A -85,B 0,C 180,E1 -7290.85,E2 -7290.85} C_VEL
LIN {X 0,Y 473.741,Z 479.349,A -85,B 0,C 180,E1 -7292.551,E2 -7292.551} C_VEL
LIN {X 0,Y 473.795,Z 477.964,A -85,B 0,C 180,E1 -7293.402,E2 -7293.402} C_VEL
LIN {X 0,Y 473.761,Z 475.039,A -85,B 0,C 180,E1 -7294.68,E2 -7294.68} C_VEL
LIN {X 0,Y 473.833,Z 471.084,A -85,B 0,C 180,E1 -7295.96,E2 -7295.96} C_VEL
LIN {X 0,Y 474.015,Z 465.012,A -85,B 0,C 180,E1 -7297.454,E2 -7297.454} C_VEL
LIN {X 0,Y 474.279,Z 458.374,A -85,B 0,C 180,E1 -7298.736,E2 -7298.736} C_VEL
LIN {X 0,Y 474.594,Z 450.139,A -85,B 0,C 180,E1 -7300.02,E2 -7300.02} C_VEL
LIN {X 0,Y 475.044,Z 441.722,A -85,B 0,C 180,E1 -7301.089,E2 -7301.089} C_VEL
LIN {X 0,Y 475.569,Z 431.548,A -85,B 0,C 180,E1 -7302.138,E2 -7302.138} C_VEL
LIN {X 0,Y 475.958,Z 419.805,A -85,B 0,C 180,E1 -7303.111,E2 -7303.111} C_VEL
LIN {X 0,Y 476.487,Z 408.038,A -85,B 0,C 180,E1 -7303.868,E2 -7303.868} C_VEL
LIN {X 0,Y 476.938,Z 395.973,A -85,B 0,C 180,E1 -7304.453,E2 -7304.453} C_VEL
LIN {X 0,Y 477.346,Z 382.866,A -85,B 0,C 180,E1 -7304.904,E2 -7304.904} C_VEL
LIN {X 0,Y 477.576,Z 370.289,A -85,B 0,C 180,E1 -7305.169,E2 -7305.169} C_VEL
LIN {X 0,Y 478.022,Z 285.186,A -85,B 0,C 180,E1 -7306.464,E2 -7306.464} C_VEL
LIN {X 0,Y 475.314,Z 268.451,A -85,B 0,C 180,E1 -7306.841,E2 -7306.841} C_VEL
LIN {X 0,Y 476.072,Z 249.977,A -85,B 0,C 180,E1 -7310.074,E2 -7310.074} C_VEL
LIN {X 0,Y 476.76,Z 233.557,A -85,B 0,C 180,E1 -7312.994,E2 -7312.994} C_VEL
LIN {X 0,Y 476.392,Z 229.007,A -85,B 0,C 180,E1 -7313.842,E2 -7313.842} C_VEL
LIN {X 0,Y 474.643,Z 220.366,A -85,B 0,C 180,E1 -7315.535,E2 -7315.535} C_VEL
LIN {X 0,Y 474.621,Z 220.365,A -85,B 0,C 180,E1 -7318.284,E2 -7318.284} C_VEL
LIN {X 0,Y 474.6,Z 220.369,A -85,B 0,C 180,E1 -7321.218,E2 -7321.218} C_VEL
LIN {X 0,Y 474.632,Z 220.36,A -85,B 0,C 180,E1 -7324.241,E2 -7324.241} C_VEL
LIN {X 0,Y 474.586,Z 220.372,A -85,B 0,C 180,E1 -7327.384,E2 -7327.384} C_VEL
LIN {X 0,Y 474.615,Z 220.362,A -85,B 0,C 180,E1 -7330.658,E2 -7330.658} C_VEL
LIN {X 0,Y 474.593,Z 220.371,A -85,B 0,C 180,E1 -7333.48,E2 -7333.48} C_VEL
LIN {X 0,Y 474.592,Z 220.364,A -85,B 0,C 180,E1 -7336.52,E2 -7336.52} C_VEL
LIN {X 0,Y 474.615,Z 220.367,A -85,B 0,C 180,E1 -7339.342,E2 -7339.342} C_VEL
LIN {X 0,Y 474.585,Z 220.363,A -85,B 0,C 180,E1 -7342.616,E2 -7342.616} C_VEL
LIN {X 0,Y 474.62,Z 220.361,A -85,B 0,C 180,E1 -7345.758,E2 -7345.758} C_VEL
LIN {X 0,Y 474.599,Z 220.363,A -85,B 0,C 180,E1 -7348.782,E2 -7348.782} C_VEL
LIN {X 0,Y 474.62,Z 220.365,A -85,B 0,C 180,E1 -7351.716,E2 -7351.716} C_VEL
LIN {X 0,Y 474.651,Z 220.353,A -85,B 0,C 180,E1 -7354.583,E2 -7354.583} C_VEL
LIN {X 0,Y 474.602,Z 220.37,A -85,B 0,C 180,E1 -7357.355,E2 -7357.355} C_VEL
LIN {X 0,Y 474.655,Z 220.356,A -85,B 0,C 180,E1 -7360.09,E2 -7360.09} C_VEL
LIN {X 0,Y 474.639,Z 220.357,A -85,B 0,C 180,E1 -7362.774,E2 -7362.774} C_VEL
LIN {X 0,Y 474.653,Z 220.363,A -85,B 0,C 180,E1 -7365.421,E2 -7365.421} C_VEL
LIN {X 0,Y 474.705,Z 220.347,A -85,B 0,C 180,E1 -7368.038,E2 -7368.038} C_VEL
LIN {X 0,Y 474.727,Z 220.351,A -85,B 0,C 180,E1 -7371.487,E2 -7371.487} C_VEL
LIN {X 0,Y 474.778,Z 220.34,A -85,B 0,C 180,E1 -7374.052,E2 -7374.052} C_VEL
LIN {X 0,Y 474.884,Z 220.33,A -85,B 0,C 180,E1 -7377.455,E2 -7377.455} C_VEL
LIN {X 0,Y 474.912,Z 220.325,A -85,B 0,C 180,E1 -7380,E2 -7380} C_VEL
LIN {X 0,Y 474.887,Z 220.324,A -85,B 0,C 180,E1 -7382.545,E2 -7382.545} C_VEL
LIN {X 0,Y 474.761,Z 220.344,A -85,B 0,C 180,E1 -7385.948,E2 -7385.948} C_VEL
LIN {X 0,Y 474.712,Z 220.344,A -85,B 0,C 180,E1 -7388.514,E2 -7388.514} C_VEL
LIN {X 0,Y 474.706,Z 220.349,A -85,B 0,C 180,E1 -7391.963,E2 -7391.963} C_VEL
